LIN {X 0,Y 498.54,Z 668.142,A -85,B 0,C 180,E1 -12477.451,E2 -12477.451} C_VEL
LIN {X 0,Y 496.811,Z 689.973,A -85,B 0,C 180,E1 -12478.358,E2 -12478.358} C_VEL
LIN {X 0,Y 494.724,Z 710.777,A -85,B 0,C 180,E1 -12479.449,E2 -12479.449} C_VEL
LIN {X 0,Y 492.444,Z 730.313,A -85,B 0,C 180,E1 -12480.703,E2 -12480.703} C_VEL
LIN {X 0,Y 489.968,Z 749.027,A -85,B 0,C 180,E1 -12482.139,E2 -12482.139} C_VEL
LIN {X 0,Y 487.302,Z 767.508,A -85,B 0,C 180,E1 -12483.822,E2 -12483.822} C_VEL
LIN {X 0,Y 484.655,Z 784.843,A -85,B 0,C 180,E1 -12485.695,E2 -12485.695} C_VEL
LIN {X 0,Y 482.176,Z 800.537,A -85,B 0,C 180,E1 -12487.698,E2 -12487.698} C_VEL
LIN {X 0,Y 479.994,Z 814.356,A -85,B 0,C 180,E1 -12489.769,E2 -12489.769} C_VEL
LIN {X 0,Y 478.09,Z 826.817,A -85,B 0,C 180,E1 -12491.969,E2 -12491.969} C_VEL
LIN {X 0,Y 476.381,Z 838.536,A -85,B 0,C 180,E1 -12494.454,E2 -12494.454} C_VEL
LIN {X 0,Y 475.075,Z 848.28,A -85,B 0,C 180,E1 -12496.985,E2 -12496.985} C_VEL
LIN {X 0,Y 474.193,Z 855.818,A -85,B 0,C 180,E1 -12499.429,E2 -12499.429} C_VEL
LIN {X 0,Y 473.59,Z 861.948,A -85,B 0,C 180,E1 -12501.99,E2 -12501.99} C_VEL
LIN {X 0,Y 473.251,Z 866.357,A -85,B 0,C 180,E1 -12504.544,E2 -12504.544} C_VEL
LIN {X 0,Y 473.077,Z 869.113,A -85,B 0,C 180,E1 -12507.092,E2 -12507.092} C_VEL
LIN {X 0,Y 473.009,Z 870.147,A -85,B 0,C 180,E1 -12509.637,E2 -12509.637} C_VEL
LIN {X 0,Y 473.046,Z 869.578,A -85,B 0,C 180,E1 -12512.18,E2 -12512.18} C_VEL
LIN {X 0,Y 473.186,Z 867.412,A -85,B 0,C 180,E1 -12514.727,E2 -12514.727} C_VEL
LIN {X 0,Y 473.468,Z 863.613,A -85,B 0,C 180,E1 -12517.279,E2 -12517.279} C_VEL
LIN {X 0,Y 473.968,Z 858.017,A -85,B 0,C 180,E1 -12519.839,E2 -12519.839} C_VEL
LIN {X 0,Y 474.756,Z 851.005,A -85,B 0,C 180,E1 -12522.282,E2 -12522.282} C_VEL
LIN {X 0,Y 475.921,Z 841.751,A -85,B 0,C 180,E1 -12524.852,E2 -12524.852} C_VEL
LIN {X 0,Y 477.437,Z 831.152,A -85,B 0,C 180,E1 -12527.254,E2 -12527.254} C_VEL
LIN {X 0,Y 479.248,Z 819.296,A -85,B 0,C 180,E1 -12529.501,E2 -12529.501} C_VEL
LIN {X 0,Y 481.426,Z 805.537,A -85,B 0,C 180,E1 -12531.697,E2 -12531.697} C_VEL
LIN {X 0,Y 483.853,Z 790.18,A -85,B 0,C 180,E1 -12533.764,E2 -12533.764} C_VEL
LIN {X 0,Y 486.381,Z 773.879,A -85,B 0,C 180,E1 -12535.625,E2 -12535.625} C_VEL
LIN {X 0,Y 488.969,Z 756.338,A -85,B 0,C 180,E1 -12537.328,E2 -12537.328} C_VEL
LIN {X 0,Y 491.47,Z 738.084,A -85,B 0,C 180,E1 -12538.827,E2 -12538.827} C_VEL
LIN {X 0,Y 493.925,Z 718.094,A -85,B 0,C 180,E1 -12540.202,E2 -12540.202} C_VEL
LIN {X 0,Y 496.061,Z 698.144,A -85,B 0,C 180,E1 -12541.335,E2 -12541.335} C_VEL
LIN {X 0,Y 497.882,Z 677.418,A -85,B 0,C 180,E1 -12542.29,E2 -12542.29} C_VEL
LIN {X 0,Y 499.402,Z 655.167,A -85,B 0,C 180,E1 -12543.082,E2 -12543.082} C_VEL
LIN {X 0,Y 501.293,Z 619.373,A -85,B 0,C 180,E1 -12543.999,E2 -12543.999} C_VEL
LIN {X 0,Y 506.162,Z 544.365,A -85,B 0,C 180,E1 -12545.618,E2 -12545.618} C_VEL
LIN {X 0,Y 509.917,Z 475.713,A -85,B 0,C 180,E1 -12546.907,E2 -12546.907} C_VEL
LIN {X 0,Y 512.618,Z 409.2,A -85,B 0,C 180,E1 -12547.977,E2 -12547.977} C_VEL
LIN {X 0,Y 513.876,Z 374.612,A -85,B 0,C 180,E1 -12548.51,E2 -12548.51} C_VEL
LIN {X 0,Y 517.445,Z 358.291,A -85,B 0,C 180,E1 -12549.153,E2 -12549.153} C_VEL
LIN {X 0,Y 517.911,Z 317.946,A -85,B 0,C 180,E1 -12551.929,E2 -12551.929} C_VEL
LIN {X 0,Y 510.317,Z 297.328,A -85,B 0,C 180,E1 -12554.386,E2 -12554.386} C_VEL
LIN {X 0,Y 502.334,Z 278.601,A -85,B 0,C 180,E1 -12556.785,E2 -12556.785} C_VEL
LIN {X 0,Y 494.836,Z 263.053,A -85,B 0,C 180,E1 -12558.95,E2 -12558.95} C_VEL
LIN {X 0,Y 487.309,Z 249.107,A -85,B 0,C 180,E1 -12561.046,E2 -12561.046} C_VEL
LIN {X 0,Y 482.169,Z 240.332,A -85,B 0,C 180,E1 -12562.434,E2 -12562.434} C_VEL
LIN {X 0,Y 479.749,Z 236.125,A -85,B 0,C 180,E1 -12563.112,E2 -12563.112} C_VEL
LIN {X 0,Y 477.498,Z 232.436,A -85,B 0,C 180,E1 -12563.726,E2 -12563.726} C_VEL
LIN {X 0,Y 476.91,Z 231.296,A -85,B 0,C 180,E1 -12563.903,E2 -12563.903} C_VEL
LIN {X 0,Y 474.742,Z 228.427,A -85,B 0,C 180,E1 -12564.457,E2 -12564.457} C_VEL
LIN {X 0,Y 474.109,Z 226.17,A -85,B 0,C 180,E1 -12564.742,E2 -12564.742} C_VEL
LIN {X 0,Y 474.113,Z 226.159,A -85,B 0,C 180,E1 -12568.464,E2 -12568.464} C_VEL
LIN {X 0,Y 474.107,Z 226.143,A -85,B 0,C 180,E1 -12572.088,E2 -12572.088} C_VEL
LIN {X 0,Y 474.108,Z 226.139,A -85,B 0,C 180,E1 -12575.716,E2 -12575.716} C_VEL
LIN {X 0,Y 474.107,Z 226.173,A -85,B 0,C 180,E1 -12579.378,E2 -12579.378} C_VEL
LIN {X 0,Y 474.105,Z 226.141,A -85,B 0,C 180,E1 -12583.08,E2 -12583.08} C_VEL
LIN {X 0,Y 474.101,Z 226.141,A -85,B 0,C 180,E1 -12586.585,E2 -12586.585} C_VEL
LIN {X 0,Y 474.099,Z 226.17,A -85,B 0,C 180,E1 -12590.286,E2 -12590.286} C_VEL
LIN {X 0,Y 474.103,Z 226.127,A -85,B 0,C 180,E1 -12593.947,E2 -12593.947} C_VEL
LIN {X 0,Y 474.112,Z 226.175,A -85,B 0,C 180,E1 -12597.583,E2 -12597.583} C_VEL
LIN {X 0,Y 474.109,Z 226.126,A -85,B 0,C 180,E1 -12601.208,E2 -12601.208} C_VEL
LIN {X 0,Y 474.1,Z 226.168,A -85,B 0,C 180,E1 -12604.839,E2 -12604.839} C_VEL
LIN {X 0,Y 474.084,Z 226.14,A -85,B 0,C 180,E1 -12608.441,E2 -12608.441} C_VEL
LIN {X 0,Y 474.099,Z 226.178,A -85,B 0,C 180,E1 -12612.052,E2 -12612.052} C_VEL
LIN {X 0,Y 474.117,Z 226.162,A -85,B 0,C 180,E1 -12615.661,E2 -12615.661} C_VEL
LIN {X 0,Y 474.116,Z 226.167,A -85,B 0,C 180,E1 -12619.336,E2 -12619.336} C_VEL
LIN {X 0,Y 474.086,Z 226.178,A -85,B 0,C 180,E1 -12622.835,E2 -12622.835} C_VEL
LIN {X 0,Y 474.083,Z 226.168,A -85,B 0,C 180,E1 -12626.425,E2 -12626.425} C_VEL
LIN {X 0,Y 474.134,Z 226.296,A -85,B 0,C 180,E1 -12627.45,E2 -12627.45} C_VEL
LIN {X 0,Y 475.326,Z 229.528,A -85,B 0,C 180,E1 -12627.976,E2 -12627.976} C_VEL
LIN {X 0,Y 476.699,Z 231.84,A -85,B 0,C 180,E1 -12628.434,E2 -12628.434} C_VEL
LIN {X 0,Y 481.647,Z 241.457,A -85,B 0,C 180,E1 -12630.158,E2 -12630.158} C_VEL
LIN {X 0,Y 489.624,Z 256.766,A -85,B 0,C 180,E1 -12632.764,E2 -12632.764} C_VEL
LIN {X 0,Y 500.094,Z 277.627,A -85,B 0,C 180,E1 -12636.003,E2 -12636.003} C_VEL
LIN {X 0,Y 511.483,Z 301.22,A -85,B 0,C 180,E1 -12639.3,E2 -12639.3} C_VEL
LIN {X 0,Y 519.807,Z 318.56,A -85,B 0,C 180,E1 -12641.486,E2 -12641.486} C_VEL
LIN {X 0,Y 522.352,Z 322.995,A -85,B 0,C 180,E1 -12641.812,E2 -12641.812} C_VEL
LIN {X 0,Y 524.642,Z 347.742,A -85,B 0,C 180,E1 -12642.536,E2 -12642.536} C_VEL
LIN {X 0,Y 513.943,Z 587.488,A -85,B 0,C 180,E1 -12646.538,E2 -12646.538} C_VEL
LIN {X 0,Y 509.832,Z 692.964,A -85,B 0,C 180,E1 -12648.278,E2 -12648.278} C_VEL
LIN {X 0,Y 508.032,Z 717.442,A -85,B 0,C 180,E1 -12648.868,E2 -12648.868} C_VEL
LIN {X 0,Y 505.864,Z 741.406,A -85,B 0,C 180,E1 -12649.63,E2 -12649.63} C_VEL
LIN {X 0,Y 503.324,Z 764.227,A -85,B 0,C 180,E1 -12650.565,E2 -12650.565} C_VEL
LIN {X 0,Y 500.285,Z 788.254,A -85,B 0,C 180,E1 -12651.764,E2 -12651.764} C_VEL
LIN {X 0,Y 497.424,Z 808.594,A -85,B 0,C 180,E1 -12652.984,E2 -12652.984} C_VEL
LIN {X 0,Y 493.885,Z 831.697,A -85,B 0,C 180,E1 -12654.618,E2 -12654.618} C_VEL
LIN {X 0,Y 490.913,Z 850.192,A -85,B 0,C 180,E1 -12656.147,E2 -12656.147} C_VEL
LIN {X 0,Y 487.599,Z 870.092,A -85,B 0,C 180,E1 -12658.058,E2 -12658.058} C_VEL
LIN {X 0,Y 484.649,Z 887.507,A -85,B 0,C 180,E1 -12659.98,E2 -12659.98} C_VEL
LIN {X 0,Y 481.773,Z 904.616,A -85,B 0,C 180,E1 -12662.162,E2 -12662.162} C_VEL
LIN {X 0,Y 479.426,Z 919.191,A -85,B 0,C 180,E1 -12664.291,E2 -12664.291} C_VEL
LIN {X 0,Y 477.164,Z 934.025,A -85,B 0,C 180,E1 -12666.799,E2 -12666.799} C_VEL
LIN {X 0,Y 475.501,Z 946.237,A -85,B 0,C 180,E1 -12669.184,E2 -12669.184} C_VEL
LIN {X 0,Y 474.103,Z 958.209,A -85,B 0,C 180,E1 -12671.939,E2 -12671.939} C_VEL
LIN {X 0,Y 473.22,Z 967.521,A -85,B 0,C 180,E1 -12674.474,E2 -12674.474} C_VEL
LIN {X 0,Y 472.64,Z 976.006,A -85,B 0,C 180,E1 -12677.29,E2 -12677.29} C_VEL
LIN {X 0,Y 472.385,Z 982.114,A -85,B 0,C 180,E1 -12679.822,E2 -12679.822} C_VEL
LIN {X 0,Y 472.289,Z 987.389,A -85,B 0,C 180,E1 -12682.702,E2 -12682.702} C_VEL
LIN {X 0,Y 472.333,Z 990.403,A -85,B 0,C 180,E1 -12685.143,E2 -12685.143} C_VEL
LIN {X 0,Y 472.382,Z 992.129,A -85,B 0,C 180,E1 -12687.452,E2 -12687.452} C_VEL
LIN {X 0,Y 472.425,Z 992.783,A -85,B 0,C 180,E1 -12690.121,E2 -12690.121} C_VEL
LIN {X 0,Y 472.4,Z 991.751,A -85,B 0,C 180,E1 -12692.79,E2 -12692.79} C_VEL
LIN {X 0,Y 472.366,Z 989.7,A -85,B 0,C 180,E1 -12695.101,E2 -12695.101} C_VEL
LIN {X 0,Y 472.343,Z 986.144,A -85,B 0,C 180,E1 -12697.664,E2 -12697.664} C_VEL
LIN {X 0,Y 472.457,Z 980.753,A -85,B 0,C 180,E1 -12700.364,E2 -12700.364} C_VEL
LIN {X 0,Y 472.711,Z 974.464,A -85,B 0,C 180,E1 -12702.832,E2 -12702.832} C_VEL
LIN {X 0,Y 473.282,Z 965.476,A -85,B 0,C 180,E1 -12705.689,E2 -12705.689} C_VEL
LIN {X 0,Y 474.142,Z 955.945,A -85,B 0,C 180,E1 -12708.186,E2 -12708.186} C_VEL
LIN {X 0,Y 475.522,Z 943.625,A -85,B 0,C 180,E1 -12710.945,E2 -12710.945} C_VEL
LIN {X 0,Y 477.241,Z 930.371,A -85,B 0,C 180,E1 -12713.458,E2 -12713.458} C_VEL
LIN {X 0,Y 479.545,Z 914.812,A -85,B 0,C 180,E1 -12716.016,E2 -12716.016} C_VEL
LIN {X 0,Y 482.006,Z 899.256,A -85,B 0,C 180,E1 -12718.227,E2 -12718.227} C_VEL
LIN {X 0,Y 485.194,Z 880.054,A -85,B 0,C 180,E1 -12720.599,E2 -12720.599} C_VEL
LIN {X 0,Y 488.36,Z 861.534,A -85,B 0,C 180,E1 -12722.58,E2 -12722.58} C_VEL
LIN {X 0,Y 491.865,Z 840.855,A -85,B 0,C 180,E1 -12724.481,E2 -12724.481} C_VEL
LIN {X 0,Y 495.389,Z 819.524,A -85,B 0,C 180,E1 -12726.177,E2 -12726.177} C_VEL
LIN {X 0,Y 498.74,Z 797.883,A -85,B 0,C 180,E1 -12727.635,E2 -12727.635} C_VEL
LIN {X 0,Y 502.253,Z 774.045,A -85,B 0,C 180,E1 -12728.984,E2 -12728.984} C_VEL
LIN {X 0,Y 505.228,Z 751.77,A -85,B 0,C 180,E1 -12730.031,E2 -12730.031} C_VEL
LIN {X 0,Y 507.919,Z 728.566,A -85,B 0,C 180,E1 -12730.907,E2 -12730.907} C_VEL
LIN {X 0,Y 510.279,Z 705.051,A -85,B 0,C 180,E1 -12731.608,E2 -12731.608} C_VEL
LIN {X 0,Y 512.094,Z 679.83,A -85,B 0,C 180,E1 -12732.154,E2 -12732.154} C_VEL
LIN {X 0,Y 517.017,Z 597.902,A -85,B 0,C 180,E1 -12733.672,E2 -12733.672} C_VEL
LIN {X 0,Y 522.642,Z 530.22,A -85,B 0,C 180,E1 -12735.047,E2 -12735.047} C_VEL
LIN {X 0,Y 529.867,Z 464.415,A -85,B 0,C 180,E1 -12736.492,E2 -12736.492} C_VEL
LIN {X 0,Y 538.765,Z 402.255,A -85,B 0,C 180,E1 -12737.913,E2 -12737.913} C_VEL
LIN {X 0,Y 544.168,Z 370.237,A -85,B 0,C 180,E1 -12738.674,E2 -12738.674} C_VEL
LIN {X 0,Y 538.418,Z 386.185,A -85,B 0,C 180,E1 -12740.242,E2 -12740.242} C_VEL
LIN {X 0,Y 534.921,Z 400.034,A -85,B 0,C 180,E1 -12741.47,E2 -12741.47} C_VEL
LIN {X 0,Y 531.61,Z 418.651,A -85,B 0,C 180,E1 -12742.928,E2 -12742.928} C_VEL
LIN {X 0,Y 528.747,Z 441.431,A -85,B 0,C 180,E1 -12744.455,E2 -12744.455} C_VEL
LIN {X 0,Y 526.309,Z 468.54,A -85,B 0,C 180,E1 -12746.028,E2 -12746.028} C_VEL
LIN {X 0,Y 524.021,Z 500.146,A -85,B 0,C 180,E1 -12747.6,E2 -12747.6} C_VEL
LIN {X 0,Y 523.085,Z 512.301,A -85,B 0,C 180,E1 -12748.121,E2 -12748.121} C_VEL
LIN {X 0,Y 507.968,Z 623.688,A -85,B 0,C 180,E1 -12751.162,E2 -12751.162} C_VEL
LIN {X 0,Y 500.211,Z 692.312,A -85,B 0,C 180,E1 -12753.095,E2 -12753.095} C_VEL
LIN {X 0,Y 497.222,Z 717.176,A -85,B 0,C 180,E1 -12754.031,E2 -12754.031} C_VEL
LIN {X 0,Y 494.515,Z 738.857,A -85,B 0,C 180,E1 -12755.066,E2 -12755.066} C_VEL
LIN {X 0,Y 491.751,Z 760.438,A -85,B 0,C 180,E1 -12756.323,E2 -12756.323} C_VEL
LIN {X 0,Y 489.036,Z 780.869,A -85,B 0,C 180,E1 -12757.774,E2 -12757.774} C_VEL
LIN {X 0,Y 486.605,Z 798.705,A -85,B 0,C 180,E1 -12759.303,E2 -12759.303} C_VEL
LIN {X 0,Y 484.482,Z 813.948,A -85,B 0,C 180,E1 -12760.843,E2 -12760.843} C_VEL
LIN {X 0,Y 482.34,Z 828.73,A -85,B 0,C 180,E1 -12762.632,E2 -12762.632} C_VEL
LIN {X 0,Y 480.502,Z 841.055,A -85,B 0,C 180,E1 -12764.428,E2 -12764.428} C_VEL
LIN {X 0,Y 478.852,Z 851.963,A -85,B 0,C 180,E1 -12766.352,E2 -12766.352} C_VEL
LIN {X 0,Y 477.393,Z 861.257,A -85,B 0,C 180,E1 -12768.4,E2 -12768.4} C_VEL
LIN {X 0,Y 476.233,Z 868.521,A -85,B 0,C 180,E1 -12770.452,E2 -12770.452} C_VEL
LIN {X 0,Y 475.29,Z 874.171,A -85,B 0,C 180,E1 -12772.627,E2 -12772.627} C_VEL
LIN {X 0,Y 474.594,Z 877.91,A -85,B 0,C 180,E1 -12774.802,E2 -12774.802} C_VEL
LIN {X 0,Y 474.097,Z 879.81,A -85,B 0,C 180,E1 -12776.978,E2 -12776.978} C_VEL
LIN {X 0,Y 473.788,Z 879.972,A -85,B 0,C 180,E1 -12779.033,E2 -12779.033} C_VEL
LIN {X 0,Y 473.605,Z 878.463,A -85,B 0,C 180,E1 -12781.21,E2 -12781.21} C_VEL
LIN {X 0,Y 473.549,Z 875.211,A -85,B 0,C 180,E1 -12783.389,E2 -12783.389} C_VEL
LIN {X 0,Y 473.645,Z 870.182,A -85,B 0,C 180,E1 -12785.573,E2 -12785.573} C_VEL
LIN {X 0,Y 473.915,Z 863.283,A -85,B 0,C 180,E1 -12787.76,E2 -12787.76} C_VEL
LIN {X 0,Y 474.405,Z 854.34,A -85,B 0,C 180,E1 -12789.952,E2 -12789.952} C_VEL
LIN {X 0,Y 475.124,Z 843.798,A -85,B 0,C 180,E1 -12792.025,E2 -12792.025} C_VEL
LIN {X 0,Y 476.057,Z 831.7,A -85,B 0,C 180,E1 -12793.983,E2 -12793.983} C_VEL
LIN {X 0,Y 477.184,Z 818.188,A -85,B 0,C 180,E1 -12795.807,E2 -12795.807} C_VEL
LIN {X 0,Y 478.539,Z 802.58,A -85,B 0,C 180,E1 -12797.574,E2 -12797.574} C_VEL
LIN {X 0,Y 480.003,Z 785.869,A -85,B 0,C 180,E1 -12799.153,E2 -12799.153} C_VEL
LIN {X 0,Y 481.552,Z 767.326,A -85,B 0,C 180,E1 -12800.607,E2 -12800.607} C_VEL
LIN {X 0,Y 483.066,Z 748.687,A -85,B 0,C 180,E1 -12801.811,E2 -12801.811} C_VEL
LIN {X 0,Y 484.603,Z 728.049,A -85,B 0,C 180,E1 -12802.888,E2 -12802.888} C_VEL
LIN {X 0,Y 486.002,Z 706.513,A -85,B 0,C 180,E1 -12803.764,E2 -12803.764} C_VEL
LIN {X 0,Y 487.201,Z 684.993,A -85,B 0,C 180,E1 -12804.407,E2 -12804.407} C_VEL
LIN {X 0,Y 491.38,Z 580.934,A -85,B 0,C 180,E1 -12806.484,E2 -12806.484} C_VEL
LIN {X 0,Y 494.767,Z 499.908,A -85,B 0,C 180,E1 -12808.079,E2 -12808.079} C_VEL
LIN {X 0,Y 489.856,Z 444.398,A -85,B 0,C 180,E1 -12809.669,E2 -12809.669} C_VEL
LIN {X 0,Y 494.577,Z 391.935,A -85,B 0,C 180,E1 -12813.597,E2 -12813.597} C_VEL
LIN {X 0,Y 499.626,Z 341.605,A -85,B 0,C 180,E1 -12817.391,E2 -12817.391} C_VEL
LIN {X 0,Y 504.089,Z 300.496,A -85,B 0,C 180,E1 -12820.518,E2 -12820.518} C_VEL
LIN {X 0,Y 497.077,Z 281.186,A -85,B 0,C 180,E1 -12822.836,E2 -12822.836} C_VEL
LIN {X 0,Y 498.864,Z 281.752,A -85,B 0,C 180,E1 -12823.116,E2 -12823.116} C_VEL
LIN {X 0,Y 503.777,Z 281.964,A -85,B 0,C 180,E1 -12823.765,E2 -12823.765} C_VEL
LIN {X 0,Y 511.406,Z 300.357,A -85,B 0,C 180,E1 -12826.095,E2 -12826.095} C_VEL
LIN {X 0,Y 517.83,Z 317.866,A -85,B 0,C 180,E1 -12828.168,E2 -12828.168} C_VEL
LIN {X 0,Y 517.363,Z 358.606,A -85,B 0,C 180,E1 -12830.97,E2 -12830.97} C_VEL
LIN {X 0,Y 513.648,Z 376.214,A -85,B 0,C 180,E1 -12831.628,E2 -12831.628} C_VEL
LIN {X 0,Y 510.519,Z 461.786,A -85,B 0,C 180,E1 -12832.95,E2 -12832.95} C_VEL
LIN {X 0,Y 507.289,Z 524.733,A -85,B 0,C 180,E1 -12834.092,E2 -12834.092} C_VEL
LIN {X 0,Y 506.039,Z 532.367,A -85,B 0,C 180,E1 -12834.17,E2 -12834.17} C_VEL
LIN {X 0,Y 499.793,Z 552.676,A -85,B 0,C 180,E1 -12834.148,E2 -12834.148} C_VEL
LIN {X 0,Y 498.777,Z 559.214,A -85,B 0,C 180,E1 -12834.234,E2 -12834.234} C_VEL
LIN {X 0,Y 493.831,Z 632.998,A -85,B 0,C 180,E1 -12835.9,E2 -12835.9} C_VEL
LIN {X 0,Y 492.338,Z 660.657,A -85,B 0,C 180,E1 -12836.672,E2 -12836.672} C_VEL
LIN {X 0,Y 490.752,Z 682.372,A -85,B 0,C 180,E1 -12837.494,E2 -12837.494} C_VEL
LIN {X 0,Y 488.846,Z 702.844,A -85,B 0,C 180,E1 -12838.481,E2 -12838.481} C_VEL
LIN {X 0,Y 486.522,Z 723.263,A -85,B 0,C 180,E1 -12839.699,E2 -12839.699} C_VEL
LIN {X 0,Y 483.983,Z 742.53,A -85,B 0,C 180,E1 -12841.09,E2 -12841.09} C_VEL
LIN {X 0,Y 481.322,Z 760.902,A -85,B 0,C 180,E1 -12842.671,E2 -12842.671} C_VEL
LIN {X 0,Y 478.596,Z 778.314,A -85,B 0,C 180,E1 -12844.442,E2 -12844.442} C_VEL
LIN {X 0,Y 476.006,Z 794.203,A -85,B 0,C 180,E1 -12846.346,E2 -12846.346} C_VEL
LIN {X 0,Y 473.532,Z 809.093,A -85,B 0,C 180,E1 -12848.444,E2 -12848.444} C_VEL
LIN {X 0,Y 471.329,Z 822.494,A -85,B 0,C 180,E1 -12850.674,E2 -12850.674} C_VEL
LIN {X 0,Y 469.449,Z 834.427,A -85,B 0,C 180,E1 -12853.034,E2 -12853.034} C_VEL
LIN {X 0,Y 467.909,Z 844.825,A -85,B 0,C 180,E1 -12855.521,E2 -12855.521} C_VEL
LIN {X 0,Y 466.793,Z 853.257,A -85,B 0,C 180,E1 -12858.008,E2 -12858.008} C_VEL
LIN {X 0,Y 466.006,Z 859.958,A -85,B 0,C 180,E1 -12860.49,E2 -12860.49} C_VEL
LIN {X 0,Y 465.509,Z 865.261,A -85,B 0,C 180,E1 -12863.091,E2 -12863.091} C_VEL
LIN {X 0,Y 465.23,Z 868.891,A -85,B 0,C 180,E1 -12865.686,E2 -12865.686} C_VEL
LIN {X 0,Y 465.099,Z 870.797,A -85,B 0,C 180,E1 -12868.275,E2 -12868.275} C_VEL
LIN {X 0,Y 465.069,Z 871.098,A -85,B 0,C 180,E1 -12870.739,E2 -12870.739} C_VEL
LIN {X 0,Y 465.149,Z 869.976,A -85,B 0,C 180,E1 -12873.204,E2 -12873.204} C_VEL
LIN {X 0,Y 465.356,Z 867.167,A -85,B 0,C 180,E1 -12875.796,E2 -12875.796} C_VEL
LIN {X 0,Y 465.713,Z 862.893,A -85,B 0,C 180,E1 -12878.271,E2 -12878.271} C_VEL
LIN {X 0,Y 466.373,Z 856.661,A -85,B 0,C 180,E1 -12880.904,E2 -12880.904} C_VEL
LIN {X 0,Y 467.313,Z 849.17,A -85,B 0,C 180,E1 -12883.361,E2 -12883.361} C_VEL
LIN {X 0,Y 468.657,Z 839.774,A -85,B 0,C 180,E1 -12885.848,E2 -12885.848} C_VEL
LIN {X 0,Y 470.425,Z 828.283,A -85,B 0,C 180,E1 -12888.335,E2 -12888.335} C_VEL
LIN {X 0,Y 472.548,Z 815.17,A -85,B 0,C 180,E1 -12890.693,E2 -12890.693} C_VEL
LIN {X 0,Y 474.847,Z 801.303,A -85,B 0,C 180,E1 -12892.796,E2 -12892.796} C_VEL
LIN {X 0,Y 477.37,Z 786.058,A -85,B 0,C 180,E1 -12894.766,E2 -12894.766} C_VEL
LIN {X 0,Y 480.042,Z 769.347,A -85,B 0,C 180,E1 -12896.604,E2 -12896.604} C_VEL
LIN {X 0,Y 482.71,Z 751.732,A -85,B 0,C 180,E1 -12898.25,E2 -12898.25} C_VEL
LIN {X 0,Y 485.282,Z 733.327,A -85,B 0,C 180,E1 -12899.705,E2 -12899.705} C_VEL
LIN {X 0,Y 487.727,Z 713.336,A -85,B 0,C 180,E1 -12901.024,E2 -12901.024} C_VEL
LIN {X 0,Y 489.988,Z 691.73,A -85,B 0,C 180,E1 -12902.182,E2 -12902.182} C_VEL
LIN {X 0,Y 491.801,Z 669.836,A -85,B 0,C 180,E1 -12903.107,E2 -12903.107} C_VEL
LIN {X 0,Y 493.107,Z 647.709,A -85,B 0,C 180,E1 -12903.816,E2 -12903.816} C_VEL
LIN {X 0,Y 495.899,Z 602.371,A -85,B 0,C 180,E1 -12904.921,E2 -12904.921} C_VEL
LIN {X 0,Y 500.552,Z 531.774,A -85,B 0,C 180,E1 -12906.421,E2 -12906.421} C_VEL
LIN {X 0,Y 504.112,Z 465.945,A -85,B 0,C 180,E1 -12907.639,E2 -12907.639} C_VEL
LIN {X 0,Y 507.201,Z 385.645,A -85,B 0,C 180,E1 -12908.901,E2 -12908.901} C_VEL
LIN {X 0,Y 507.596,Z 377.376,A -85,B 0,C 180,E1 -12909.04,E2 -12909.04} C_VEL
LIN {X 0,Y 511.408,Z 359.689,A -85,B 0,C 180,E1 -12909.743,E2 -12909.743} C_VEL
LIN {X 0,Y 511.798,Z 321.583,A -85,B 0,C 180,E1 -12912.378,E2 -12912.378} C_VEL
LIN {X 0,Y 503.702,Z 299.721,A -85,B 0,C 180,E1 -12915.033,E2 -12915.033} C_VEL
LIN {X 0,Y 495.259,Z 280.206,A -85,B 0,C 180,E1 -12917.598,E2 -12917.598} C_VEL
LIN {X 0,Y 487.022,Z 263.522,A -85,B 0,C 180,E1 -12920.013,E2 -12920.013} C_VEL
LIN {X 0,Y 480.126,Z 251.024,A -85,B 0,C 180,E1 -12921.943,E2 -12921.943} C_VEL
LIN {X 0,Y 474.875,Z 242.046,A -85,B 0,C 180,E1 -12923.424,E2 -12923.424} C_VEL
LIN {X 0,Y 472.072,Z 237.344,A -85,B 0,C 180,E1 -12924.226,E2 -12924.226} C_VEL
LIN {X 0,Y 469.994,Z 234.244,A -85,B 0,C 180,E1 -12924.792,E2 -12924.792} C_VEL
LIN {X 0,Y 469.308,Z 232.581,A -85,B 0,C 180,E1 -12925.032,E2 -12925.032} C_VEL
LIN {X 0,Y 467.108,Z 230.042,A -85,B 0,C 180,E1 -12925.589,E2 -12925.589} C_VEL
LIN {X 0,Y 466.171,Z 227.144,A -85,B 0,C 180,E1 -12925.994,E2 -12925.994} C_VEL
LIN {X 0,Y 466.183,Z 227.157,A -85,B 0,C 180,E1 -12929.732,E2 -12929.732} C_VEL
LIN {X 0,Y 466.167,Z 227.157,A -85,B 0,C 180,E1 -12933.435,E2 -12933.435} C_VEL
LIN {X 0,Y 466.163,Z 227.125,A -85,B 0,C 180,E1 -12937.155,E2 -12937.155} C_VEL
LIN {X 0,Y 466.169,Z 227.13,A -85,B 0,C 180,E1 -12940.712,E2 -12940.712} C_VEL
LIN {X 0,Y 466.166,Z 227.16,A -85,B 0,C 180,E1 -12944.448,E2 -12944.448} C_VEL
LIN {X 0,Y 466.157,Z 227.117,A -85,B 0,C 180,E1 -12948.117,E2 -12948.117} C_VEL
LIN {X 0,Y 466.173,Z 227.152,A -85,B 0,C 180,E1 -12951.737,E2 -12951.737} C_VEL
LIN {X 0,Y 466.167,Z 227.131,A -85,B 0,C 180,E1 -12955.448,E2 -12955.448} C_VEL
LIN {X 0,Y 466.172,Z 227.129,A -85,B 0,C 180,E1 -12959.14,E2 -12959.14} C_VEL
LIN {X 0,Y 466.16,Z 227.153,A -85,B 0,C 180,E1 -12962.828,E2 -12962.828} C_VEL
LIN {X 0,Y 466.145,Z 227.119,A -85,B 0,C 180,E1 -12966.404,E2 -12966.404} C_VEL
LIN {X 0,Y 466.16,Z 227.164,A -85,B 0,C 180,E1 -12970.09,E2 -12970.09} C_VEL
LIN {X 0,Y 466.178,Z 227.164,A -85,B 0,C 180,E1 -12973.773,E2 -12973.773} C_VEL
LIN {X 0,Y 466.178,Z 227.161,A -85,B 0,C 180,E1 -12977.475,E2 -12977.475} C_VEL
LIN {X 0,Y 466.164,Z 227.154,A -85,B 0,C 180,E1 -12981.122,E2 -12981.122} C_VEL
LIN {X 0,Y 466.143,Z 227.158,A -85,B 0,C 180,E1 -12984.726,E2 -12984.726} C_VEL
LIN {X 0,Y 466.167,Z 227.306,A -85,B 0,C 180,E1 -12986.359,E2 -12986.359} C_VEL
LIN {X 0,Y 467.547,Z 230.773,A -85,B 0,C 180,E1 -12986.961,E2 -12986.961} C_VEL
LIN {X 0,Y 468.637,Z 232.398,A -85,B 0,C 180,E1 -12987.305,E2 -12987.305} C_VEL
LIN {X 0,Y 470.585,Z 236.188,A -85,B 0,C 180,E1 -12988.007,E2 -12988.007} C_VEL
LIN {X 0,Y 479.969,Z 254.318,A -85,B 0,C 180,E1 -12991.247,E2 -12991.247} C_VEL
LIN {X 0,Y 490.555,Z 275.349,A -85,B 0,C 180,E1 -12994.659,E2 -12994.659} C_VEL
LIN {X 0,Y 500.946,Z 296.719,A -85,B 0,C 180,E1 -12997.791,E2 -12997.791} C_VEL
LIN {X 0,Y 511.695,Z 319.213,A -85,B 0,C 180,E1 -13000.761,E2 -13000.761} C_VEL
LIN {X 0,Y 516.358,Z 326.875,A -85,B 0,C 180,E1 -13001.352,E2 -13001.352} C_VEL
LIN {X 0,Y 518.336,Z 348.872,A -85,B 0,C 180,E1 -13002.004,E2 -13002.004} C_VEL
LIN {X 0,Y 507.238,Z 586.374,A -85,B 0,C 180,E1 -13006.036,E2 -13006.036} C_VEL
LIN {X 0,Y 502.902,Z 692.911,A -85,B 0,C 180,E1 -13007.824,E2 -13007.824} C_VEL
LIN {X 0,Y 501.042,Z 717.485,A -85,B 0,C 180,E1 -13008.425,E2 -13008.425} C_VEL
LIN {X 0,Y 498.81,Z 741.363,A -85,B 0,C 180,E1 -13009.195,E2 -13009.195} C_VEL
LIN {X 0,Y 496.263,Z 763.656,A -85,B 0,C 180,E1 -13010.117,E2 -13010.117} C_VEL
LIN {X 0,Y 493.243,Z 787.052,A -85,B 0,C 180,E1 -13011.29,E2 -13011.29} C_VEL
LIN {X 0,Y 490.284,Z 807.507,A -85,B 0,C 180,E1 -13012.525,E2 -13012.525} C_VEL
LIN {X 0,Y 486.843,Z 829.512,A -85,B 0,C 180,E1 -13014.085,E2 -13014.085} C_VEL
LIN {X 0,Y 483.717,Z 848.3,A -85,B 0,C 180,E1 -13015.645,E2 -13015.645} C_VEL
LIN {X 0,Y 480.169,Z 869.073,A -85,B 0,C 180,E1 -13017.645,E2 -13017.645} C_VEL
LIN {X 0,Y 477.21,Z 886.031,A -85,B 0,C 180,E1 -13019.532,E2 -13019.532} C_VEL
LIN {X 0,Y 474.101,Z 903.893,A -85,B 0,C 180,E1 -13021.833,E2 -13021.833} C_VEL
LIN {X 0,Y 471.568,Z 919.187,A -85,B 0,C 180,E1 -13024.101,E2 -13024.101} C_VEL
LIN {X 0,Y 469.349,Z 933.266,A -85,B 0,C 180,E1 -13026.523,E2 -13026.523} C_VEL
LIN {X 0,Y 467.629,Z 945.482,A -85,B 0,C 180,E1 -13028.948,E2 -13028.948} C_VEL
LIN {X 0,Y 466.173,Z 957.477,A -85,B 0,C 180,E1 -13031.751,E2 -13031.751} C_VEL
LIN {X 0,Y 465.263,Z 966.781,A -85,B 0,C 180,E1 -13034.322,E2 -13034.322} C_VEL
LIN {X 0,Y 464.669,Z 975.278,A -85,B 0,C 180,E1 -13037.195,E2 -13037.195} C_VEL
LIN {X 0,Y 464.416,Z 981.244,A -85,B 0,C 180,E1 -13039.714,E2 -13039.714} C_VEL
LIN {X 0,Y 464.32,Z 986.433,A -85,B 0,C 180,E1 -13042.576,E2 -13042.576} C_VEL
LIN {X 0,Y 464.373,Z 989.471,A -85,B 0,C 180,E1 -13045.059,E2 -13045.059} C_VEL
LIN {X 0,Y 464.429,Z 991.213,A -85,B 0,C 180,E1 -13047.409,E2 -13047.409} C_VEL
LIN {X 0,Y 464.477,Z 991.875,A -85,B 0,C 180,E1 -13050.123,E2 -13050.123} C_VEL
LIN {X 0,Y 464.447,Z 990.846,A -85,B 0,C 180,E1 -13052.838,E2 -13052.838} C_VEL
LIN {X 0,Y 464.405,Z 988.778,A -85,B 0,C 180,E1 -13055.188,E2 -13055.188} C_VEL
LIN {X 0,Y 464.382,Z 985.207,A -85,B 0,C 180,E1 -13057.796,E2 -13057.796} C_VEL
LIN {X 0,Y 464.483,Z 979.801,A -85,B 0,C 180,E1 -13060.543,E2 -13060.543} C_VEL
LIN {X 0,Y 464.771,Z 973.134,A -85,B 0,C 180,E1 -13063.182,E2 -13063.182} C_VEL
LIN {X 0,Y 465.389,Z 964.01,A -85,B 0,C 180,E1 -13066.091,E2 -13066.091} C_VEL
LIN {X 0,Y 466.305,Z 954.396,A -85,B 0,C 180,E1 -13068.633,E2 -13068.633} C_VEL
LIN {X 0,Y 467.802,Z 941.928,A -85,B 0,C 180,E1 -13071.438,E2 -13071.438} C_VEL
LIN {X 0,Y 469.561,Z 929.295,A -85,B 0,C 180,E1 -13073.865,E2 -13073.865} C_VEL
LIN {X 0,Y 471.941,Z 914.029,A -85,B 0,C 180,E1 -13076.418,E2 -13076.418} C_VEL
LIN {X 0,Y 474.607,Z 898.182,A -85,B 0,C 180,E1 -13078.708,E2 -13078.708} C_VEL
LIN {X 0,Y 477.963,Z 879.004,A -85,B 0,C 180,E1 -13081.113,E2 -13081.113} C_VEL
LIN {X 0,Y 481.406,Z 860.028,A -85,B 0,C 180,E1 -13083.171,E2 -13083.171} C_VEL
LIN {X 0,Y 485.017,Z 839.842,A -85,B 0,C 180,E1 -13085.047,E2 -13085.047} C_VEL
LIN {X 0,Y 488.706,Z 818.705,A -85,B 0,C 180,E1 -13086.753,E2 -13086.753} C_VEL
LIN {X 0,Y 492.221,Z 797.381,A -85,B 0,C 180,E1 -13088.211,E2 -13088.211} C_VEL
LIN {X 0,Y 495.94,Z 773.646,A -85,B 0,C 180,E1 -13089.576,E2 -13089.576} C_VEL
LIN {X 0,Y 499.069,Z 751.686,A -85,B 0,C 180,E1 -13090.628,E2 -13090.628} C_VEL
LIN {X 0,Y 501.964,Z 728.472,A -85,B 0,C 180,E1 -13091.523,E2 -13091.523} C_VEL
LIN {X 0,Y 504.399,Z 706.193,A -85,B 0,C 180,E1 -13092.208,E2 -13092.208} C_VEL
LIN {X 0,Y 506.382,Z 681.601,A -85,B 0,C 180,E1 -13092.767,E2 -13092.767} C_VEL
LIN {X 0,Y 511.96,Z 599.732,A -85,B 0,C 180,E1 -13094.343,E2 -13094.343} C_VEL
LIN {X 0,Y 518.163,Z 533.367,A -85,B 0,C 180,E1 -13095.738,E2 -13095.738} C_VEL
LIN {X 0,Y 525.811,Z 470.913,A -85,B 0,C 180,E1 -13097.15,E2 -13097.15} C_VEL
LIN {X 0,Y 535.086,Z 411.727,A -85,B 0,C 180,E1 -13098.528,E2 -13098.528} C_VEL
LIN {X 0,Y 539.64,Z 386.423,A -85,B 0,C 180,E1 -13099.133,E2 -13099.133} C_VEL
LIN {X 0,Y 534.431,Z 402.446,A -85,B 0,C 180,E1 -13100.59,E2 -13100.59} C_VEL
LIN {X 0,Y 530.546,Z 419.16,A -85,B 0,C 180,E1 -13101.938,E2 -13101.938} C_VEL
LIN {X 0,Y 526.896,Z 440.675,A -85,B 0,C 180,E1 -13103.45,E2 -13103.45} C_VEL
LIN {X 0,Y 523.592,Z 467.503,A -85,B 0,C 180,E1 -13105.072,E2 -13105.072} C_VEL
LIN {X 0,Y 520.576,Z 498.689,A -85,B 0,C 180,E1 -13106.687,E2 -13106.687} C_VEL
LIN {X 0,Y 519.163,Z 513.949,A -85,B 0,C 180,E1 -13107.374,E2 -13107.374} C_VEL
LIN {X 0,Y 503.179,Z 623.523,A -85,B 0,C 180,E1 -13110.425,E2 -13110.425} C_VEL
LIN {X 0,Y 494.715,Z 692.559,A -85,B 0,C 180,E1 -13112.421,E2 -13112.421} C_VEL
LIN {X 0,Y 491.531,Z 716.722,A -85,B 0,C 180,E1 -13113.349,E2 -13113.349} C_VEL
LIN {X 0,Y 488.391,Z 739.771,A -85,B 0,C 180,E1 -13114.471,E2 -13114.471} C_VEL
LIN {X 0,Y 485.547,Z 760.078,A -85,B 0,C 180,E1 -13115.678,E2 -13115.678} C_VEL
LIN {X 0,Y 482.62,Z 780.56,A -85,B 0,C 180,E1 -13117.141,E2 -13117.141} C_VEL
LIN {X 0,Y 479.706,Z 800.352,A -85,B 0,C 180,E1 -13118.863,E2 -13118.863} C_VEL
LIN {X 0,Y 477.171,Z 816.917,A -85,B 0,C 180,E1 -13120.602,E2 -13120.602} C_VEL
LIN {X 0,Y 475.127,Z 830.018,A -85,B 0,C 180,E1 -13122.233,E2 -13122.233} C_VEL
LIN {X 0,Y 473.167,Z 842.333,A -85,B 0,C 180,E1 -13124.055,E2 -13124.055} C_VEL
LIN {X 0,Y 471.382,Z 853.157,A -85,B 0,C 180,E1 -13126.006,E2 -13126.006} C_VEL
LIN {X 0,Y 469.813,Z 862.453,A -85,B 0,C 180,E1 -13128.086,E2 -13128.086} C_VEL
LIN {X 0,Y 468.488,Z 870.052,A -85,B 0,C 180,E1 -13130.293,E2 -13130.293} C_VEL
LIN {X 0,Y 467.481,Z 875.602,A -85,B 0,C 180,E1 -13132.503,E2 -13132.503} C_VEL
LIN {X 0,Y 466.732,Z 879.228,A -85,B 0,C 180,E1 -13134.714,E2 -13134.714} C_VEL
LIN {X 0,Y 466.2,Z 881.03,A -85,B 0,C 180,E1 -13136.926,E2 -13136.926} C_VEL
LIN {X 0,Y 465.854,Z 881.048,A -85,B 0,C 180,E1 -13139.139,E2 -13139.139} C_VEL
LIN {X 0,Y 465.66,Z 879.31,A -85,B 0,C 180,E1 -13141.353,E2 -13141.353} C_VEL
LIN {X 0,Y 465.608,Z 875.845,A -85,B 0,C 180,E1 -13143.571,E2 -13143.571} C_VEL
LIN {X 0,Y 465.719,Z 870.596,A -85,B 0,C 180,E1 -13145.792,E2 -13145.792} C_VEL
LIN {X 0,Y 466.015,Z 863.458,A -85,B 0,C 180,E1 -13148.017,E2 -13148.017} C_VEL
LIN {X 0,Y 466.507,Z 854.813,A -85,B 0,C 180,E1 -13150.123,E2 -13150.123} C_VEL
LIN {X 0,Y 467.208,Z 844.805,A -85,B 0,C 180,E1 -13152.107,E2 -13152.107} C_VEL
LIN {X 0,Y 468.166,Z 832.719,A -85,B 0,C 180,E1 -13154.092,E2 -13154.092} C_VEL
LIN {X 0,Y 469.327,Z 819.151,A -85,B 0,C 180,E1 -13155.952,E2 -13155.952} C_VEL
LIN {X 0,Y 470.666,Z 804.108,A -85,B 0,C 180,E1 -13157.686,E2 -13157.686} C_VEL
LIN {X 0,Y 472.163,Z 787.528,A -85,B 0,C 180,E1 -13159.291,E2 -13159.291} C_VEL
LIN {X 0,Y 473.767,Z 769.076,A -85,B 0,C 180,E1 -13160.779,E2 -13160.779} C_VEL
LIN {X 0,Y 475.377,Z 749.813,A -85,B 0,C 180,E1 -13162.052,E2 -13162.052} C_VEL
LIN {X 0,Y 476.956,Z 729.338,A -85,B 0,C 180,E1 -13163.146,E2 -13163.146} C_VEL
LIN {X 0,Y 478.443,Z 707.237,A -85,B 0,C 180,E1 -13164.066,E2 -13164.066} C_VEL
LIN {X 0,Y 479.691,Z 685.63,A -85,B 0,C 180,E1 -13164.729,E2 -13164.729} C_VEL
LIN {X 0,Y 481.691,Z 636.241,A -85,B 0,C 180,E1 -13165.753,E2 -13165.753} C_VEL
LIN {X 0,Y 487.592,Z 500.852,A -85,B 0,C 180,E1 -13168.482,E2 -13168.482} C_VEL
LIN {X 0,Y 482.649,Z 443.526,A -85,B 0,C 180,E1 -13170.158,E2 -13170.158} C_VEL
LIN {X 0,Y 487.555,Z 391.321,A -85,B 0,C 180,E1 -13174.114,E2 -13174.114} C_VEL
LIN {X 0,Y 492.883,Z 340.388,A -85,B 0,C 180,E1 -13178.003,E2 -13178.003} C_VEL
LIN {X 0,Y 497.018,Z 303.388,A -85,B 0,C 180,E1 -13180.849,E2 -13180.849} C_VEL
LIN {X 0,Y 491.675,Z 288.4,A -85,B 0,C 180,E1 -13182.665,E2 -13182.665} C_VEL
LIN {X 0,Y 493.95,Z 288.989,A -85,B 0,C 180,E1 -13183.015,E2 -13183.015} C_VEL
LIN {X 0,Y 499.293,Z 289.309,A -85,B 0,C 180,E1 -13183.741,E2 -13183.741} C_VEL
LIN {X 0,Y 507.081,Z 308.783,A -85,B 0,C 180,E1 -13186.202,E2 -13186.202} C_VEL
LIN {X 0,Y 511.777,Z 322.105,A -85,B 0,C 180,E1 -13187.772,E2 -13187.772} C_VEL
LIN {X 0,Y 511.313,Z 360.22,A -85,B 0,C 180,E1 -13190.398,E2 -13190.398} C_VEL
LIN {X 0,Y 507.373,Z 378.886,A -85,B 0,C 180,E1 -13191.096,E2 -13191.096} C_VEL
LIN {X 0,Y 504.154,Z 463.908,A -85,B 0,C 180,E1 -13192.422,E2 -13192.422} C_VEL
LIN {X 0,Y 500.507,Z 531.887,A -85,B 0,C 180,E1 -13193.677,E2 -13193.677} C_VEL
LIN {X 0,Y 498.777,Z 559.214,A -85,B 0,C 180,E1 -13194.234,E2 -13194.234} C_VEL
LIN {X 0,Y 497.486,Z 566.831,A -85,B 0,C 180,E1 -13194.326,E2 -13194.326} C_VEL
LIN {X 0,Y 491.089,Z 587.097,A -85,B 0,C 180,E1 -13194.33,E2 -13194.33} C_VEL
LIN {X 0,Y 490.025,Z 593.617,A -85,B 0,C 180,E1 -13194.426,E2 -13194.426} C_VEL
LIN {X 0,Y 486.575,Z 645.419,A -85,B 0,C 180,E1 -13195.686,E2 -13195.686} C_VEL
LIN {X 0,Y 485.245,Z 667.881,A -85,B 0,C 180,E1 -13196.386,E2 -13196.386} C_VEL
LIN {X 0,Y 483.547,Z 688.635,A -85,B 0,C 180,E1 -13197.239,E2 -13197.239} C_VEL
LIN {X 0,Y 481.427,Z 709.184,A -85,B 0,C 180,E1 -13198.3,E2 -13198.3} C_VEL
LIN {X 0,Y 478.958,Z 729.358,A -85,B 0,C 180,E1 -13199.578,E2 -13199.578} C_VEL
LIN {X 0,Y 476.375,Z 747.976,A -85,B 0,C 180,E1 -13200.997,E2 -13200.997} C_VEL
LIN {X 0,Y 473.544,Z 766.359,A -85,B 0,C 180,E1 -13202.661,E2 -13202.661} C_VEL
LIN {X 0,Y 470.669,Z 783.837,A -85,B 0,C 180,E1 -13204.539,E2 -13204.539} C_VEL
LIN {X 0,Y 467.905,Z 799.872,A -85,B 0,C 180,E1 -13206.58,E2 -13206.58} C_VEL
LIN {X 0,Y 465.271,Z 814.963,A -85,B 0,C 180,E1 -13208.858,E2 -13208.858} C_VEL
LIN {X 0,Y 463.008,Z 828.125,A -85,B 0,C 180,E1 -13211.23,E2 -13211.23} C_VEL
LIN {X 0,Y 461.172,Z 839.251,A -85,B 0,C 180,E1 -13213.629,E2 -13213.629} C_VEL
LIN {X 0,Y 459.702,Z 848.945,A -85,B 0,C 180,E1 -13216.157,E2 -13216.157} C_VEL
LIN {X 0,Y 458.578,Z 857.298,A -85,B 0,C 180,E1 -13218.87,E2 -13218.87} C_VEL
LIN {X 0,Y 457.875,Z 863.459,A -85,B 0,C 180,E1 -13221.46,E2 -13221.46} C_VEL
LIN {X 0,Y 457.457,Z 868.051,A -85,B 0,C 180,E1 -13224.103,E2 -13224.103} C_VEL
LIN {X 0,Y 457.224,Z 870.89,A -85,B 0,C 180,E1 -13226.74,E2 -13226.74} C_VEL
LIN {X 0,Y 457.135,Z 872.082,A -85,B 0,C 180,E1 -13229.248,E2 -13229.248} C_VEL
LIN {X 0,Y 457.162,Z 871.849,A -85,B 0,C 180,E1 -13231.755,E2 -13231.755} C_VEL
LIN {X 0,Y 457.302,Z 869.964,A -85,B 0,C 180,E1 -13234.403,E2 -13234.403} C_VEL
LIN {X 0,Y 457.597,Z 866.416,A -85,B 0,C 180,E1 -13237.029,E2 -13237.029} C_VEL
LIN {X 0,Y 458.118,Z 861.185,A -85,B 0,C 180,E1 -13239.675,E2 -13239.675} C_VEL
LIN {X 0,Y 458.958,Z 854.552,A -85,B 0,C 180,E1 -13242.2,E2 -13242.2} C_VEL
LIN {X 0,Y 460.152,Z 846.045,A -85,B 0,C 180,E1 -13244.767,E2 -13244.767} C_VEL
LIN {X 0,Y 461.846,Z 835.297,A -85,B 0,C 180,E1 -13247.384,E2 -13247.384} C_VEL
LIN {X 0,Y 463.962,Z 822.671,A -85,B 0,C 180,E1 -13249.908,E2 -13249.908} C_VEL
LIN {X 0,Y 466.31,Z 809.091,A -85,B 0,C 180,E1 -13252.172,E2 -13252.172} C_VEL
LIN {X 0,Y 468.767,Z 794.94,A -85,B 0,C 180,E1 -13254.176,E2 -13254.176} C_VEL
LIN {X 0,Y 471.488,Z 778.982,A -85,B 0,C 180,E1 -13256.107,E2 -13256.107} C_VEL
LIN {X 0,Y 474.336,Z 761.484,A -85,B 0,C 180,E1 -13257.903,E2 -13257.903} C_VEL
LIN {X 0,Y 477.008,Z 743.797,A -85,B 0,C 180,E1 -13259.443,E2 -13259.443} C_VEL
LIN {X 0,Y 479.644,Z 724.54,A -85,B 0,C 180,E1 -13260.852,E2 -13260.852} C_VEL
LIN {X 0,Y 482.044,Z 704.365,A -85,B 0,C 180,E1 -13262.074,E2 -13262.074} C_VEL
LIN {X 0,Y 484.165,Z 682.397,A -85,B 0,C 180,E1 -13263.145,E2 -13263.145} C_VEL
LIN {X 0,Y 485.877,Z 659.344,A -85,B 0,C 180,E1 -13264.008,E2 -13264.008} C_VEL
LIN {X 0,Y 487.914,Z 623.727,A -85,B 0,C 180,E1 -13264.967,E2 -13264.967} C_VEL
LIN {X 0,Y 492.911,Z 552.333,A -85,B 0,C 180,E1 -13266.57,E2 -13266.57} C_VEL
LIN {X 0,Y 496.796,Z 487.533,A -85,B 0,C 180,E1 -13267.835,E2 -13267.835} C_VEL
LIN {X 0,Y 499.705,Z 423.65,A -85,B 0,C 180,E1 -13268.904,E2 -13268.904} C_VEL
LIN {X 0,Y 501.36,Z 380.151,A -85,B 0,C 180,E1 -13269.583,E2 -13269.583} C_VEL
LIN {X 0,Y 505.415,Z 361.597,A -85,B 0,C 180,E1 -13270.31,E2 -13270.31} C_VEL
LIN {X 0,Y 505.768,Z 325.409,A -85,B 0,C 180,E1 -13272.823,E2 -13272.823} C_VEL
LIN {X 0,Y 497.877,Z 304.182,A -85,B 0,C 180,E1 -13275.42,E2 -13275.42} C_VEL
LIN {X 0,Y 489.767,Z 285.201,A -85,B 0,C 180,E1 -13277.961,E2 -13277.961} C_VEL
LIN {X 0,Y 481.64,Z 268.543,A -85,B 0,C 180,E1 -13280.406,E2 -13280.406} C_VEL
LIN {X 0,Y 474.838,Z 256.177,A -85,B 0,C 180,E1 -13282.362,E2 -13282.362} C_VEL
LIN {X 0,Y 470.082,Z 247.938,A -85,B 0,C 180,E1 -13283.749,E2 -13283.749} C_VEL
LIN {X 0,Y 467.272,Z 243.314,A -85,B 0,C 180,E1 -13284.556,E2 -13284.556} C_VEL
LIN {X 0,Y 464.53,Z 238.712,A -85,B 0,C 180,E1 -13285.371,E2 -13285.371} C_VEL
LIN {X 0,Y 462.104,Z 235.133,A -85,B 0,C 180,E1 -13286.065,E2 -13286.065} C_VEL
LIN {X 0,Y 461.413,Z 233.57,A -85,B 0,C 180,E1 -13286.306,E2 -13286.306} C_VEL
LIN {X 0,Y 459.273,Z 231.197,A -85,B 0,C 180,E1 -13286.876,E2 -13286.876} C_VEL
LIN {X 0,Y 458.221,Z 228.122,A -85,B 0,C 180,E1 -13287.311,E2 -13287.311} C_VEL
LIN {X 0,Y 458.227,Z 228.119,A -85,B 0,C 180,E1 -13291.047,E2 -13291.047} C_VEL
LIN {X 0,Y 458.232,Z 228.139,A -85,B 0,C 180,E1 -13294.679,E2 -13294.679} C_VEL
LIN {X 0,Y 458.229,Z 228.136,A -85,B 0,C 180,E1 -13298.367,E2 -13298.367} C_VEL
LIN {X 0,Y 458.225,Z 228.105,A -85,B 0,C 180,E1 -13302.081,E2 -13302.081} C_VEL
LIN {X 0,Y 458.235,Z 228.133,A -85,B 0,C 180,E1 -13305.854,E2 -13305.854} C_VEL
LIN {X 0,Y 458.231,Z 228.13,A -85,B 0,C 180,E1 -13309.565,E2 -13309.565} C_VEL
LIN {X 0,Y 458.23,Z 228.107,A -85,B 0,C 180,E1 -13313.233,E2 -13313.233} C_VEL
LIN {X 0,Y 458.23,Z 228.15,A -85,B 0,C 180,E1 -13316.998,E2 -13316.998} C_VEL
LIN {X 0,Y 458.214,Z 228.1,A -85,B 0,C 180,E1 -13320.625,E2 -13320.625} C_VEL
LIN {X 0,Y 458.213,Z 228.15,A -85,B 0,C 180,E1 -13324.38,E2 -13324.38} C_VEL
LIN {X 0,Y 458.218,Z 228.106,A -85,B 0,C 180,E1 -13328.028,E2 -13328.028} C_VEL
LIN {X 0,Y 458.234,Z 228.151,A -85,B 0,C 180,E1 -13331.708,E2 -13331.708} C_VEL
LIN {X 0,Y 458.242,Z 228.138,A -85,B 0,C 180,E1 -13335.439,E2 -13335.439} C_VEL
LIN {X 0,Y 458.227,Z 228.143,A -85,B 0,C 180,E1 -13339.118,E2 -13339.118} C_VEL
LIN {X 0,Y 458.206,Z 228.157,A -85,B 0,C 180,E1 -13342.721,E2 -13342.721} C_VEL
LIN {X 0,Y 458.248,Z 228.309,A -85,B 0,C 180,E1 -13345.216,E2 -13345.216} C_VEL
LIN {X 0,Y 459.502,Z 231.574,A -85,B 0,C 180,E1 -13345.799,E2 -13345.799} C_VEL
LIN {X 0,Y 460.611,Z 233.05,A -85,B 0,C 180,E1 -13346.147,E2 -13346.147} C_VEL
LIN {X 0,Y 462.422,Z 236.877,A -85,B 0,C 180,E1 -13346.867,E2 -13346.867} C_VEL
LIN {X 0,Y 470.046,Z 251.38,A -85,B 0,C 180,E1 -13349.572,E2 -13349.572} C_VEL
LIN {X 0,Y 479.662,Z 270.434,A -85,B 0,C 180,E1 -13352.819,E2 -13352.819} C_VEL
LIN {X 0,Y 489.067,Z 289.421,A -85,B 0,C 180,E1 -13355.784,E2 -13355.784} C_VEL
LIN {X 0,Y 499.32,Z 310.731,A -85,B 0,C 180,E1 -13358.813,E2 -13358.813} C_VEL
LIN {X 0,Y 504.05,Z 320.505,A -85,B 0,C 180,E1 -13360.07,E2 -13360.07} C_VEL
LIN {X 0,Y 510.322,Z 330.764,A -85,B 0,C 180,E1 -13360.894,E2 -13360.894} C_VEL
LIN {X 0,Y 511.985,Z 350.164,A -85,B 0,C 180,E1 -13361.474,E2 -13361.474} C_VEL
LIN {X 0,Y 500.204,Z 594.045,A -85,B 0,C 180,E1 -13365.667,E2 -13365.667} C_VEL
LIN {X 0,Y 495.978,Z 693.246,A -85,B 0,C 180,E1 -13367.366,E2 -13367.366} C_VEL
LIN {X 0,Y 494.054,Z 717.678,A -85,B 0,C 180,E1 -13367.976,E2 -13367.976} C_VEL
LIN {X 0,Y 491.76,Z 741.384,A -85,B 0,C 180,E1 -13368.754,E2 -13368.754} C_VEL
LIN {X 0,Y 489.157,Z 763.478,A -85,B 0,C 180,E1 -13369.681,E2 -13369.681} C_VEL
LIN {X 0,Y 486.107,Z 786.461,A -85,B 0,C 180,E1 -13370.847,E2 -13370.847} C_VEL
LIN {X 0,Y 482.946,Z 807.676,A -85,B 0,C 180,E1 -13372.146,E2 -13372.146} C_VEL
LIN {X 0,Y 479.236,Z 830.66,A -85,B 0,C 180,E1 -13373.81,E2 -13373.81} C_VEL
LIN {X 0,Y 475.951,Z 849.917,A -85,B 0,C 180,E1 -13375.443,E2 -13375.443} C_VEL
LIN {X 0,Y 472.486,Z 869.477,A -85,B 0,C 180,E1 -13377.38,E2 -13377.38} C_VEL
LIN {X 0,Y 469.3,Z 887.249,A -85,B 0,C 180,E1 -13379.403,E2 -13379.403} C_VEL
LIN {X 0,Y 466.342,Z 903.708,A -85,B 0,C 180,E1 -13381.576,E2 -13381.576} C_VEL
LIN {X 0,Y 463.846,Z 918.314,A -85,B 0,C 180,E1 -13383.774,E2 -13383.774} C_VEL
LIN {X 0,Y 461.437,Z 933.109,A -85,B 0,C 180,E1 -13386.367,E2 -13386.367} C_VEL
LIN {X 0,Y 459.594,Z 945.92,A -85,B 0,C 180,E1 -13388.963,E2 -13388.963} C_VEL
LIN {X 0,Y 458.192,Z 957.214,A -85,B 0,C 180,E1 -13391.685,E2 -13391.685} C_VEL
LIN {X 0,Y 457.245,Z 966.776,A -85,B 0,C 180,E1 -13394.397,E2 -13394.397} C_VEL
LIN {X 0,Y 456.681,Z 974.841,A -85,B 0,C 180,E1 -13397.224,E2 -13397.224} C_VEL
LIN {X 0,Y 456.438,Z 980.733,A -85,B 0,C 180,E1 -13399.779,E2 -13399.779} C_VEL
LIN {X 0,Y 456.363,Z 985.805,A -85,B 0,C 180,E1 -13402.699,E2 -13402.699} C_VEL
LIN {X 0,Y 456.421,Z 988.645,A -85,B 0,C 180,E1 -13405.099,E2 -13405.099} C_VEL
LIN {X 0,Y 456.484,Z 990.35,A -85,B 0,C 180,E1 -13407.489,E2 -13407.489} C_VEL
LIN {X 0,Y 456.52,Z 990.948,A -85,B 0,C 180,E1 -13410.251,E2 -13410.251} C_VEL
LIN {X 0,Y 456.496,Z 989.935,A -85,B 0,C 180,E1 -13412.888,E2 -13412.888} C_VEL
LIN {X 0,Y 456.445,Z 987.861,A -85,B 0,C 180,E1 -13415.279,E2 -13415.279} C_VEL
LIN {X 0,Y 456.426,Z 984.128,A -85,B 0,C 180,E1 -13418.028,E2 -13418.028} C_VEL
LIN {X 0,Y 456.512,Z 978.559,A -85,B 0,C 180,E1 -13420.857,E2 -13420.857} C_VEL
LIN {X 0,Y 456.806,Z 972.154,A -85,B 0,C 180,E1 -13423.416,E2 -13423.416} C_VEL
LIN {X 0,Y 457.471,Z 963.024,A -85,B 0,C 180,E1 -13426.377,E2 -13426.377} C_VEL
LIN {X 0,Y 458.432,Z 953.388,A -85,B 0,C 180,E1 -13428.965,E2 -13428.965} C_VEL
LIN {X 0,Y 460.047,Z 940.686,A -85,B 0,C 180,E1 -13431.864,E2 -13431.864} C_VEL
LIN {X 0,Y 461.929,Z 928.114,A -85,B 0,C 180,E1 -13434.314,E2 -13434.314} C_VEL
LIN {X 0,Y 464.561,Z 912.168,A -85,B 0,C 180,E1 -13437.01,E2 -13437.01} C_VEL
LIN {X 0,Y 467.24,Z 897.186,A -85,B 0,C 180,E1 -13439.204,E2 -13439.204} C_VEL
LIN {X 0,Y 470.791,Z 878.062,A -85,B 0,C 180,E1 -13441.641,E2 -13441.641} C_VEL
LIN {X 0,Y 474.441,Z 859.063,A -85,B 0,C 180,E1 -13443.734,E2 -13443.734} C_VEL
LIN {X 0,Y 478.199,Z 839.149,A -85,B 0,C 180,E1 -13445.615,E2 -13445.615} C_VEL
LIN {X 0,Y 482.12,Z 818.027,A -85,B 0,C 180,E1 -13447.346,E2 -13447.346} C_VEL
LIN {X 0,Y 485.785,Z 797.142,A -85,B 0,C 180,E1 -13448.798,E2 -13448.798} C_VEL
LIN {X 0,Y 489.724,Z 773.628,A -85,B 0,C 180,E1 -13450.18,E2 -13450.18} C_VEL
LIN {X 0,Y 493.009,Z 752.05,A -85,B 0,C 180,E1 -13451.235,E2 -13451.235} C_VEL
LIN {X 0,Y 496.262,Z 727.875,A -85,B 0,C 180,E1 -13452.189,E2 -13452.189} C_VEL
LIN {X 0,Y 498.951,Z 704.878,A -85,B 0,C 180,E1 -13452.906,E2 -13452.906} C_VEL
LIN {X 0,Y 501.206,Z 679.012,A -85,B 0,C 180,E1 -13453.498,E2 -13453.498} C_VEL
LIN {X 0,Y 506.91,Z 604.456,A -85,B 0,C 180,E1 -13454.984,E2 -13454.984} C_VEL
LIN {X 0,Y 513.515,Z 540.682,A -85,B 0,C 180,E1 -13456.364,E2 -13456.364} C_VEL
LIN {X 0,Y 521.895,Z 478.411,A -85,B 0,C 180,E1 -13457.804,E2 -13457.804} C_VEL
LIN {X 0,Y 532.261,Z 418.01,A -85,B 0,C 180,E1 -13459.232,E2 -13459.232} C_VEL
LIN {X 0,Y 535.068,Z 403.51,A -85,B 0,C 180,E1 -13459.593,E2 -13459.593} C_VEL
LIN {X 0,Y 529.965,Z 420.849,A -85,B 0,C 180,E1 -13461.024,E2 -13461.024} C_VEL
LIN {X 0,Y 525.36,Z 442.234,A -85,B 0,C 180,E1 -13462.56,E2 -13462.56} C_VEL
LIN {X 0,Y 521.359,Z 467.462,A -85,B 0,C 180,E1 -13464.133,E2 -13464.133} C_VEL
LIN {X 0,Y 517.712,Z 496.915,A -85,B 0,C 180,E1 -13465.72,E2 -13465.72} C_VEL
LIN {X 0,Y 515.606,Z 515.721,A -85,B 0,C 180,E1 -13466.602,E2 -13466.602} C_VEL
LIN {X 0,Y 498.716,Z 623.519,A -85,B 0,C 180,E1 -13469.657,E2 -13469.657} C_VEL
LIN {X 0,Y 489.462,Z 693.045,A -85,B 0,C 180,E1 -13471.718,E2 -13471.718} C_VEL
LIN {X 0,Y 485.921,Z 717.566,A -85,B 0,C 180,E1 -13472.686,E2 -13472.686} C_VEL
LIN {X 0,Y 482.406,Z 741.177,A -85,B 0,C 180,E1 -13473.867,E2 -13473.867} C_VEL
LIN {X 0,Y 479.01,Z 763.375,A -85,B 0,C 180,E1 -13475.234,E2 -13475.234} C_VEL
LIN {X 0,Y 475.96,Z 782.652,A -85,B 0,C 180,E1 -13476.672,E2 -13476.672} C_VEL
LIN {X 0,Y 473.172,Z 800.284,A -85,B 0,C 180,E1 -13478.231,E2 -13478.231} C_VEL
LIN {X 0,Y 470.431,Z 816.956,A -85,B 0,C 180,E1 -13479.989,E2 -13479.989} C_VEL
LIN {X 0,Y 467.973,Z 831.456,A -85,B 0,C 180,E1 -13481.823,E2 -13481.823} C_VEL
LIN {X 0,Y 465.858,Z 843.626,A -85,B 0,C 180,E1 -13483.67,E2 -13483.67} C_VEL
LIN {X 0,Y 463.953,Z 854.446,A -85,B 0,C 180,E1 -13485.65,E2 -13485.65} C_VEL
LIN {X 0,Y 462.258,Z 863.686,A -85,B 0,C 180,E1 -13487.762,E2 -13487.762} C_VEL
LIN {X 0,Y 460.893,Z 870.899,A -85,B 0,C 180,E1 -13489.879,E2 -13489.879} C_VEL
LIN {X 0,Y 459.777,Z 876.529,A -85,B 0,C 180,E1 -13492.125,E2 -13492.125} C_VEL
LIN {X 0,Y 458.985,Z 880.06,A -85,B 0,C 180,E1 -13494.249,E2 -13494.249} C_VEL
LIN {X 0,Y 458.376,Z 882.037,A -85,B 0,C 180,E1 -13496.498,E2 -13496.498} C_VEL
LIN {X 0,Y 457.98,Z 882.254,A -85,B 0,C 180,E1 -13498.749,E2 -13498.749} C_VEL
LIN {X 0,Y 457.742,Z 880.699,A -85,B 0,C 180,E1 -13501.001,E2 -13501.001} C_VEL
LIN {X 0,Y 457.661,Z 877.402,A -85,B 0,C 180,E1 -13503.256,E2 -13503.256} C_VEL
LIN {X 0,Y 457.746,Z 872.332,A -85,B 0,C 180,E1 -13505.515,E2 -13505.515} C_VEL
LIN {X 0,Y 458.022,Z 865.378,A -85,B 0,C 180,E1 -13507.779,E2 -13507.779} C_VEL
LIN {X 0,Y 458.534,Z 856.372,A -85,B 0,C 180,E1 -13510.047,E2 -13510.047} C_VEL
LIN {X 0,Y 459.29,Z 845.771,A -85,B 0,C 180,E1 -13512.191,E2 -13512.191} C_VEL
LIN {X 0,Y 460.275,Z 833.663,A -85,B 0,C 180,E1 -13514.21,E2 -13514.21} C_VEL
LIN {X 0,Y 461.471,Z 820.087,A -85,B 0,C 180,E1 -13516.102,E2 -13516.102} C_VEL
LIN {X 0,Y 462.908,Z 804.481,A -85,B 0,C 180,E1 -13517.927,E2 -13517.927} C_VEL
LIN {X 0,Y 464.458,Z 787.813,A -85,B 0,C 180,E1 -13519.558,E2 -13519.558} C_VEL
LIN {X 0,Y 466.117,Z 769.248,A -85,B 0,C 180,E1 -13521.07,E2 -13521.07} C_VEL
LIN {X 0,Y 467.783,Z 749.889,A -85,B 0,C 180,E1 -13522.363,E2 -13522.363} C_VEL
LIN {X 0,Y 469.412,Z 729.333,A -85,B 0,C 180,E1 -13523.474,E2 -13523.474} C_VEL
LIN {X 0,Y 470.946,Z 707.195,A -85,B 0,C 180,E1 -13524.407,E2 -13524.407} C_VEL
LIN {X 0,Y 472.25,Z 685.306,A -85,B 0,C 180,E1 -13525.087,E2 -13525.087} C_VEL
LIN {X 0,Y 476.139,Z 594.578,A -85,B 0,C 180,E1 -13526.978,E2 -13526.978} C_VEL
LIN {X 0,Y 480.399,Z 501.629,A -85,B 0,C 180,E1 -13528.893,E2 -13528.893} C_VEL
LIN {X 0,Y 475.428,Z 442.959,A -85,B 0,C 180,E1 -13530.633,E2 -13530.633} C_VEL
LIN {X 0,Y 480.616,Z 390.245,A -85,B 0,C 180,E1 -13534.681,E2 -13534.681} C_VEL
LIN {X 0,Y 486.158,Z 339.219,A -85,B 0,C 180,E1 -13538.625,E2 -13538.625} C_VEL
LIN {X 0,Y 489.964,Z 306.282,A -85,B 0,C 180,E1 -13541.19,E2 -13541.19} C_VEL
LIN {X 0,Y 486.224,Z 295.751,A -85,B 0,C 180,E1 -13542.488,E2 -13542.488} C_VEL
LIN {X 0,Y 488.357,Z 296.309,A -85,B 0,C 180,E1 -13542.825,E2 -13542.825} C_VEL
LIN {X 0,Y 494.683,Z 296.459,A -85,B 0,C 180,E1 -13543.691,E2 -13543.691} C_VEL
LIN {X 0,Y 502.56,Z 316.624,A -85,B 0,C 180,E1 -13546.239,E2 -13546.239} C_VEL
LIN {X 0,Y 505.822,Z 326.064,A -85,B 0,C 180,E1 -13547.338,E2 -13547.338} C_VEL
LIN {X 0,Y 505.293,Z 362.094,A -85,B 0,C 180,E1 -13549.827,E2 -13549.827} C_VEL
LIN {X 0,Y 501.139,Z 381.657,A -85,B 0,C 180,E1 -13550.552,E2 -13550.552} C_VEL
LIN {X 0,Y 497.822,Z 466.245,A -85,B 0,C 180,E1 -13551.885,E2 -13551.885} C_VEL
LIN {X 0,Y 494.1,Z 533.338,A -85,B 0,C 180,E1 -13553.138,E2 -13553.138} C_VEL
LIN {X 0,Y 490.025,Z 593.617,A -85,B 0,C 180,E1 -13554.426,E2 -13554.426} C_VEL
LIN {X 0,Y 488.675,Z 601.21,A -85,B 0,C 180,E1 -13554.531,E2 -13554.531} C_VEL
LIN {X 0,Y 482.152,Z 621.424,A -85,B 0,C 180,E1 -13554.569,E2 -13554.569} C_VEL
LIN {X 0,Y 481.085,Z 627.928,A -85,B 0,C 180,E1 -13554.677,E2 -13554.677} C_VEL
LIN {X 0,Y 479.076,Z 661.98,A -85,B 0,C 180,E1 -13555.628,E2 -13555.628} C_VEL
LIN {X 0,Y 477.368,Z 684.08,A -85,B 0,C 180,E1 -13556.476,E2 -13556.476} C_VEL
LIN {X 0,Y 475.188,Z 705.766,A -85,B 0,C 180,E1 -13557.549,E2 -13557.549} C_VEL
LIN {X 0,Y 472.71,Z 725.9,A -85,B 0,C 180,E1 -13558.786,E2 -13558.786} C_VEL
LIN {X 0,Y 469.934,Z 745.461,A -85,B 0,C 180,E1 -13560.241,E2 -13560.241} C_VEL
LIN {X 0,Y 467.104,Z 763.42,A -85,B 0,C 180,E1 -13561.835,E2 -13561.835} C_VEL
LIN {X 0,Y 464.147,Z 780.829,A -85,B 0,C 180,E1 -13563.66,E2 -13563.66} C_VEL
LIN {X 0,Y 461.249,Z 797.096,A -85,B 0,C 180,E1 -13565.677,E2 -13565.677} C_VEL
LIN {X 0,Y 458.555,Z 811.859,A -85,B 0,C 180,E1 -13567.838,E2 -13567.838} C_VEL
LIN {X 0,Y 456.146,Z 825.154,A -85,B 0,C 180,E1 -13570.137,E2 -13570.137} C_VEL
LIN {X 0,Y 454.078,Z 836.979,A -85,B 0,C 180,E1 -13572.574,E2 -13572.574} C_VEL
LIN {X 0,Y 452.378,Z 847.3,A -85,B 0,C 180,E1 -13575.144,E2 -13575.144} C_VEL
LIN {X 0,Y 451.083,Z 856.031,A -85,B 0,C 180,E1 -13577.843,E2 -13577.843} C_VEL
LIN {X 0,Y 450.214,Z 862.595,A -85,B 0,C 180,E1 -13580.434,E2 -13580.434} C_VEL
LIN {X 0,Y 449.668,Z 867.666,A -85,B 0,C 180,E1 -13583.103,E2 -13583.103} C_VEL
LIN {X 0,Y 449.371,Z 871.007,A -85,B 0,C 180,E1 -13585.661,E2 -13585.661} C_VEL
LIN {X 0,Y 449.224,Z 872.865,A -85,B 0,C 180,E1 -13588.342,E2 -13588.342} C_VEL
LIN {X 0,Y 449.198,Z 873.077,A -85,B 0,C 180,E1 -13590.893,E2 -13590.893} C_VEL
LIN {X 0,Y 449.3,Z 871.752,A -85,B 0,C 180,E1 -13593.572,E2 -13593.572} C_VEL
LIN {X 0,Y 449.556,Z 868.955,A -85,B 0,C 180,E1 -13596.168,E2 -13596.168} C_VEL
LIN {X 0,Y 450.042,Z 864.162,A -85,B 0,C 180,E1 -13598.947,E2 -13598.947} C_VEL
LIN {X 0,Y 450.791,Z 858.057,A -85,B 0,C 180,E1 -13601.515,E2 -13601.515} C_VEL
LIN {X 0,Y 451.971,Z 849.84,A -85,B 0,C 180,E1 -13604.215,E2 -13604.215} C_VEL
LIN {X 0,Y 453.537,Z 840.114,A -85,B 0,C 180,E1 -13606.787,E2 -13606.787} C_VEL
LIN {X 0,Y 455.484,Z 828.952,A -85,B 0,C 180,E1 -13609.225,E2 -13609.225} C_VEL
LIN {X 0,Y 457.768,Z 816.401,A -85,B 0,C 180,E1 -13611.528,E2 -13611.528} C_VEL
LIN {X 0,Y 460.491,Z 801.535,A -85,B 0,C 180,E1 -13613.82,E2 -13613.82} C_VEL
LIN {X 0,Y 463.393,Z 785.44,A -85,B 0,C 180,E1 -13615.909,E2 -13615.909} C_VEL
LIN {X 0,Y 466.333,Z 768.344,A -85,B 0,C 180,E1 -13617.784,E2 -13617.784} C_VEL
LIN {X 0,Y 469.068,Z 751.399,A -85,B 0,C 180,E1 -13619.359,E2 -13619.359} C_VEL
LIN {X 0,Y 471.842,Z 732.449,A -85,B 0,C 180,E1 -13620.852,E2 -13620.852} C_VEL
LIN {X 0,Y 474.38,Z 712.797,A -85,B 0,C 180,E1 -13622.142,E2 -13622.142} C_VEL
LIN {X 0,Y 476.62,Z 692.451,A -85,B 0,C 180,E1 -13623.235,E2 -13623.235} C_VEL
LIN {X 0,Y 478.464,Z 671.503,A -85,B 0,C 180,E1 -13624.133,E2 -13624.133} C_VEL
LIN {X 0,Y 479.862,Z 649.328,A -85,B 0,C 180,E1 -13624.856,E2 -13624.856} C_VEL
LIN {X 0,Y 482.942,Z 603.252,A -85,B 0,C 180,E1 -13626.015,E2 -13626.015} C_VEL
LIN {X 0,Y 487.734,Z 535.64,A -85,B 0,C 180,E1 -13627.496,E2 -13627.496} C_VEL
LIN {X 0,Y 491.458,Z 471.348,A -85,B 0,C 180,E1 -13628.716,E2 -13628.716} C_VEL
LIN {X 0,Y 494.698,Z 393.121,A -85,B 0,C 180,E1 -13629.971,E2 -13629.971} C_VEL
LIN {X 0,Y 495.169,Z 382.888,A -85,B 0,C 180,E1 -13630.14,E2 -13630.14} C_VEL
LIN {X 0,Y 499.455,Z 363.438,A -85,B 0,C 180,E1 -13630.892,E2 -13630.892} C_VEL
LIN {X 0,Y 499.819,Z 329.349,A -85,B 0,C 180,E1 -13633.265,E2 -13633.265} C_VEL
LIN {X 0,Y 492.328,Z 309.141,A -85,B 0,C 180,E1 -13635.763,E2 -13635.763} C_VEL
LIN {X 0,Y 484.713,Z 291.025,A -85,B 0,C 180,E1 -13638.218,E2 -13638.218} C_VEL
LIN {X 0,Y 477.071,Z 275.122,A -85,B 0,C 180,E1 -13640.576,E2 -13640.576} C_VEL
LIN {X 0,Y 470.415,Z 262.693,A -85,B 0,C 180,E1 -13642.561,E2 -13642.561} C_VEL
LIN {X 0,Y 464.9,Z 253.177,A -85,B 0,C 180,E1 -13644.196,E2 -13644.196} C_VEL
LIN {X 0,Y 462.135,Z 248.659,A -85,B 0,C 180,E1 -13645.015,E2 -13645.015} C_VEL
LIN {X 0,Y 459.823,Z 244.742,A -85,B 0,C 180,E1 -13645.722,E2 -13645.722} C_VEL
LIN {X 0,Y 457.513,Z 240.985,A -85,B 0,C 180,E1 -13646.432,E2 -13646.432} C_VEL
LIN {X 0,Y 456.303,Z 239.305,A -85,B 0,C 180,E1 -13646.782,E2 -13646.782} C_VEL
LIN {X 0,Y 454.022,Z 235.539,A -85,B 0,C 180,E1 -13647.496,E2 -13647.496} C_VEL
LIN {X 0,Y 453.254,Z 234.387,A -85,B 0,C 180,E1 -13647.733,E2 -13647.733} C_VEL
LIN {X 0,Y 451.199,Z 231.945,A -85,B 0,C 180,E1 -13648.317,E2 -13648.317} C_VEL
LIN {X 0,Y 450.296,Z 229.13,A -85,B 0,C 180,E1 -13648.748,E2 -13648.748} C_VEL
LIN {X 0,Y 450.293,Z 229.11,A -85,B 0,C 180,E1 -13652.492,E2 -13652.492} C_VEL
LIN {X 0,Y 450.286,Z 229.098,A -85,B 0,C 180,E1 -13656.188,E2 -13656.188} C_VEL
LIN {X 0,Y 450.291,Z 229.127,A -85,B 0,C 180,E1 -13659.933,E2 -13659.933} C_VEL
LIN {X 0,Y 450.291,Z 229.116,A -85,B 0,C 180,E1 -13663.62,E2 -13663.62} C_VEL
LIN {X 0,Y 450.288,Z 229.092,A -85,B 0,C 180,E1 -13667.301,E2 -13667.301} C_VEL
LIN {X 0,Y 450.295,Z 229.139,A -85,B 0,C 180,E1 -13671.058,E2 -13671.058} C_VEL
LIN {X 0,Y 450.283,Z 229.094,A -85,B 0,C 180,E1 -13674.776,E2 -13674.776} C_VEL
LIN {X 0,Y 450.278,Z 229.126,A -85,B 0,C 180,E1 -13678.473,E2 -13678.473} C_VEL
LIN {X 0,Y 450.274,Z 229.113,A -85,B 0,C 180,E1 -13682.291,E2 -13682.291} C_VEL
LIN {X 0,Y 450.283,Z 229.099,A -85,B 0,C 180,E1 -13685.991,E2 -13685.991} C_VEL
LIN {X 0,Y 450.294,Z 229.133,A -85,B 0,C 180,E1 -13689.716,E2 -13689.716} C_VEL
LIN {X 0,Y 450.3,Z 229.139,A -85,B 0,C 180,E1 -13693.483,E2 -13693.483} C_VEL
LIN {X 0,Y 450.292,Z 229.142,A -85,B 0,C 180,E1 -13697.177,E2 -13697.177} C_VEL
LIN {X 0,Y 450.271,Z 229.136,A -85,B 0,C 180,E1 -13700.812,E2 -13700.812} C_VEL
LIN {X 0,Y 450.313,Z 229.351,A -85,B 0,C 180,E1 -13704.066,E2 -13704.066} C_VEL
LIN {X 0,Y 451.415,Z 232.38,A -85,B 0,C 180,E1 -13704.609,E2 -13704.609} C_VEL
LIN {X 0,Y 452.816,Z 234.512,A -85,B 0,C 180,E1 -13705.085,E2 -13705.085} C_VEL
LIN {X 0,Y 460.155,Z 248.689,A -85,B 0,C 180,E1 -13707.852,E2 -13707.852} C_VEL
LIN {X 0,Y 468.901,Z 265.678,A -85,B 0,C 180,E1 -13710.925,E2 -13710.925} C_VEL
LIN {X 0,Y 478.993,Z 285.851,A -85,B 0,C 180,E1 -13714.245,E2 -13714.245} C_VEL
LIN {X 0,Y 489.169,Z 306.954,A -85,B 0,C 180,E1 -13717.379,E2 -13717.379} C_VEL
LIN {X 0,Y 496.135,Z 321.396,A -85,B 0,C 180,E1 -13719.333,E2 -13719.333} C_VEL
LIN {X 0,Y 504.323,Z 334.524,A -85,B 0,C 180,E1 -13720.418,E2 -13720.418} C_VEL
LIN {X 0,Y 505.676,Z 351.379,A -85,B 0,C 180,E1 -13720.93,E2 -13720.93} C_VEL
LIN {X 0,Y 493.439,Z 594.424,A -85,B 0,C 180,E1 -13725.177,E2 -13725.177} C_VEL
LIN {X 0,Y 489.052,Z 693.147,A -85,B 0,C 180,E1 -13726.899,E2 -13726.899} C_VEL
LIN {X 0,Y 487.064,Z 717.705,A -85,B 0,C 180,E1 -13727.52,E2 -13727.52} C_VEL
LIN {X 0,Y 484.689,Z 741.475,A -85,B 0,C 180,E1 -13728.313,E2 -13728.313} C_VEL
LIN {X 0,Y 482.008,Z 763.641,A -85,B 0,C 180,E1 -13729.256,E2 -13729.256} C_VEL
LIN {X 0,Y 478.771,Z 787.263,A -85,B 0,C 180,E1 -13730.479,E2 -13730.479} C_VEL
LIN {X 0,Y 475.64,Z 807.713,A -85,B 0,C 180,E1 -13731.75,E2 -13731.75} C_VEL
LIN {X 0,Y 471.802,Z 830.773,A -85,B 0,C 180,E1 -13733.45,E2 -13733.45} C_VEL
LIN {X 0,Y 468.306,Z 850.667,A -85,B 0,C 180,E1 -13735.17,E2 -13735.17} C_VEL
LIN {X 0,Y 464.826,Z 869.705,A -85,B 0,C 180,E1 -13737.096,E2 -13737.096} C_VEL
LIN {X 0,Y 461.569,Z 887.432,A -85,B 0,C 180,E1 -13739.147,E2 -13739.147} C_VEL
LIN {X 0,Y 458.56,Z 903.615,A -85,B 0,C 180,E1 -13741.334,E2 -13741.334} C_VEL
LIN {X 0,Y 455.749,Z 919.662,A -85,B 0,C 180,E1 -13743.809,E2 -13743.809} C_VEL
LIN {X 0,Y 453.421,Z 933.611,A -85,B 0,C 180,E1 -13746.338,E2 -13746.338} C_VEL
LIN {X 0,Y 451.558,Z 946.259,A -85,B 0,C 180,E1 -13748.979,E2 -13748.979} C_VEL
LIN {X 0,Y 450.159,Z 957.389,A -85,B 0,C 180,E1 -13751.749,E2 -13751.749} C_VEL
LIN {X 0,Y 449.189,Z 967.193,A -85,B 0,C 180,E1 -13754.639,E2 -13754.639} C_VEL
LIN {X 0,Y 448.675,Z 974.712,A -85,B 0,C 180,E1 -13757.385,E2 -13757.385} C_VEL
LIN {X 0,Y 448.445,Z 981.014,A -85,B 0,C 180,E1 -13760.244,E2 -13760.244} C_VEL
LIN {X 0,Y 448.43,Z 985.494,A -85,B 0,C 180,E1 -13763.084,E2 -13763.084} C_VEL
LIN {X 0,Y 448.492,Z 988.15,A -85,B 0,C 180,E1 -13765.525,E2 -13765.525} C_VEL
LIN {X 0,Y 448.566,Z 989.821,A -85,B 0,C 180,E1 -13768.34,E2 -13768.34} C_VEL
LIN {X 0,Y 448.582,Z 989.831,A -85,B 0,C 180,E1 -13771.022,E2 -13771.022} C_VEL
LIN {X 0,Y 448.552,Z 988.674,A -85,B 0,C 180,E1 -13773.451,E2 -13773.451} C_VEL
LIN {X 0,Y 448.472,Z 985.962,A -85,B 0,C 180,E1 -13776.272,E2 -13776.272} C_VEL
LIN {X 0,Y 448.462,Z 981.519,A -85,B 0,C 180,E1 -13779.108,E2 -13779.108} C_VEL
LIN {X 0,Y 448.59,Z 976.15,A -85,B 0,C 180,E1 -13781.703,E2 -13781.703} C_VEL
LIN {X 0,Y 449.049,Z 968.252,A -85,B 0,C 180,E1 -13784.705,E2 -13784.705} C_VEL
LIN {X 0,Y 449.779,Z 959.77,A -85,B 0,C 180,E1 -13787.331,E2 -13787.331} C_VEL
LIN {X 0,Y 451.063,Z 948.711,A -85,B 0,C 180,E1 -13790.231,E2 -13790.231} C_VEL
LIN {X 0,Y 452.845,Z 936.106,A -85,B 0,C 180,E1 -13793.006,E2 -13793.006} C_VEL
LIN {X 0,Y 455.38,Z 920.711,A -85,B 0,C 180,E1 -13795.91,E2 -13795.91} C_VEL
LIN {X 0,Y 458.179,Z 905.313,A -85,B 0,C 180,E1 -13798.408,E2 -13798.408} C_VEL
LIN {X 0,Y 461.612,Z 887.583,A -85,B 0,C 180,E1 -13800.888,E2 -13800.888} C_VEL
LIN {X 0,Y 465.255,Z 869.575,A -85,B 0,C 180,E1 -13803.085,E2 -13803.085} C_VEL
LIN {X 0,Y 469.16,Z 850.023,A -85,B 0,C 180,E1 -13805.13,E2 -13805.13} C_VEL
LIN {X 0,Y 473.357,Z 829.218,A -85,B 0,C 180,E1 -13807.016,E2 -13807.016} C_VEL
LIN {X 0,Y 477.469,Z 807.865,A -85,B 0,C 180,E1 -13808.669,E2 -13808.669} C_VEL
LIN {X 0,Y 481.578,Z 785.351,A -85,B 0,C 180,E1 -13810.142,E2 -13810.142} C_VEL
LIN {X 0,Y 485.477,Z 762.75,A -85,B 0,C 180,E1 -13811.387,E2 -13811.387} C_VEL
LIN {X 0,Y 489.041,Z 739.355,A -85,B 0,C 180,E1 -13812.432,E2 -13812.432} C_VEL
LIN {X 0,Y 492.468,Z 713.955,A -85,B 0,C 180,E1 -13813.33,E2 -13813.33} C_VEL
LIN {X 0,Y 495.235,Z 689.22,A -85,B 0,C 180,E1 -13813.991,E2 -13813.991} C_VEL
LIN {X 0,Y 502.415,Z 606.101,A -85,B 0,C 180,E1 -13815.717,E2 -13815.717} C_VEL
LIN {X 0,Y 509.652,Z 543.883,A -85,B 0,C 180,E1 -13817.107,E2 -13817.107} C_VEL
LIN {X 0,Y 518.608,Z 484.008,A -85,B 0,C 180,E1 -13818.523,E2 -13818.523} C_VEL
LIN {X 0,Y 529.824,Z 424.254,A -85,B 0,C 180,E1 -13819.952,E2 -13819.952} C_VEL
LIN {X 0,Y 530.345,Z 421.728,A -85,B 0,C 180,E1 -13820.022,E2 -13820.022} C_VEL
LIN {X 0,Y 525.481,Z 439.424,A -85,B 0,C 180,E1 -13821.347,E2 -13821.347} C_VEL
LIN {X 0,Y 521.194,Z 459.651,A -85,B 0,C 180,E1 -13822.691,E2 -13822.691} C_VEL
LIN {X 0,Y 517.046,Z 484.385,A -85,B 0,C 180,E1 -13824.138,E2 -13824.138} C_VEL
LIN {X 0,Y 512.915,Z 514.472,A -85,B 0,C 180,E1 -13825.684,E2 -13825.684} C_VEL
LIN {X 0,Y 511.601,Z 522.309,A -85,B 0,C 180,E1 -13825.939,E2 -13825.939} C_VEL
LIN {X 0,Y 494.044,Z 627.424,A -85,B 0,C 180,E1 -13828.967,E2 -13828.967} C_VEL
LIN {X 0,Y 484.529,Z 693.436,A -85,B 0,C 180,E1 -13830.974,E2 -13830.974} C_VEL
LIN {X 0,Y 480.673,Z 717.867,A -85,B 0,C 180,E1 -13831.958,E2 -13831.958} C_VEL
LIN {X 0,Y 476.883,Z 740.991,A -85,B 0,C 180,E1 -13833.138,E2 -13833.138} C_VEL
LIN {X 0,Y 473.152,Z 763.244,A -85,B 0,C 180,E1 -13834.529,E2 -13834.529} C_VEL
LIN {X 0,Y 469.661,Z 783.67,A -85,B 0,C 180,E1 -13836.073,E2 -13836.073} C_VEL
LIN {X 0,Y 466.419,Z 802.263,A -85,B 0,C 180,E1 -13837.767,E2 -13837.767} C_VEL
LIN {X 0,Y 463.679,Z 817.604,A -85,B 0,C 180,E1 -13839.421,E2 -13839.421} C_VEL
LIN {X 0,Y 461.038,Z 832.136,A -85,B 0,C 180,E1 -13841.278,E2 -13841.278} C_VEL
LIN {X 0,Y 458.61,Z 845.081,A -85,B 0,C 180,E1 -13843.274,E2 -13843.274} C_VEL
LIN {X 0,Y 456.552,Z 855.769,A -85,B 0,C 180,E1 -13845.283,E2 -13845.283} C_VEL
LIN {X 0,Y 454.829,Z 864.486,A -85,B 0,C 180,E1 -13847.3,E2 -13847.3} C_VEL
LIN {X 0,Y 453.255,Z 872.152,A -85,B 0,C 180,E1 -13849.578,E2 -13849.578} C_VEL
LIN {X 0,Y 452.041,Z 877.742,A -85,B 0,C 180,E1 -13851.862,E2 -13851.862} C_VEL
LIN {X 0,Y 451.139,Z 881.424,A -85,B 0,C 180,E1 -13854.148,E2 -13854.148} C_VEL
LIN {X 0,Y 450.515,Z 883.217,A -85,B 0,C 180,E1 -13856.31,E2 -13856.31} C_VEL
LIN {X 0,Y 450.074,Z 883.39,A -85,B 0,C 180,E1 -13858.6,E2 -13858.6} C_VEL
LIN {X 0,Y 449.815,Z 881.823,A -85,B 0,C 180,E1 -13860.892,E2 -13860.892} C_VEL
LIN {X 0,Y 449.716,Z 878.498,A -85,B 0,C 180,E1 -13863.186,E2 -13863.186} C_VEL
LIN {X 0,Y 449.795,Z 873.387,A -85,B 0,C 180,E1 -13865.485,E2 -13865.485} C_VEL
LIN {X 0,Y 450.067,Z 866.52,A -85,B 0,C 180,E1 -13867.753,E2 -13867.753} C_VEL
LIN {X 0,Y 450.558,Z 857.917,A -85,B 0,C 180,E1 -13869.968,E2 -13869.968} C_VEL
LIN {X 0,Y 451.318,Z 847.405,A -85,B 0,C 180,E1 -13872.15,E2 -13872.15} C_VEL
LIN {X 0,Y 452.311,Z 835.396,A -85,B 0,C 180,E1 -13874.204,E2 -13874.204} C_VEL
LIN {X 0,Y 453.613,Z 820.956,A -85,B 0,C 180,E1 -13876.257,E2 -13876.257} C_VEL
LIN {X 0,Y 455.089,Z 805.309,A -85,B 0,C 180,E1 -13878.113,E2 -13878.113} C_VEL
LIN {X 0,Y 456.753,Z 787.953,A -85,B 0,C 180,E1 -13879.835,E2 -13879.835} C_VEL
LIN {X 0,Y 458.462,Z 769.351,A -85,B 0,C 180,E1 -13881.365,E2 -13881.365} C_VEL
LIN {X 0,Y 460.196,Z 749.84,A -85,B 0,C 180,E1 -13882.685,E2 -13882.685} C_VEL
LIN {X 0,Y 461.88,Z 729.249,A -85,B 0,C 180,E1 -13883.812,E2 -13883.812} C_VEL
LIN {X 0,Y 463.467,Z 707.122,A -85,B 0,C 180,E1 -13884.76,E2 -13884.76} C_VEL
LIN {X 0,Y 464.819,Z 685.119,A -85,B 0,C 180,E1 -13885.452,E2 -13885.452} C_VEL
LIN {X 0,Y 473.257,Z 502.713,A -85,B 0,C 180,E1 -13889.308,E2 -13889.308} C_VEL
LIN {X 0,Y 468.265,Z 442.042,A -85,B 0,C 180,E1 -13891.15,E2 -13891.15} C_VEL
LIN {X 0,Y 473.624,Z 389.762,A -85,B 0,C 180,E1 -13895.213,E2 -13895.213} C_VEL
LIN {X 0,Y 479.379,Z 338.841,A -85,B 0,C 180,E1 -13899.198,E2 -13899.198} C_VEL
LIN {X 0,Y 482.929,Z 309.227,A -85,B 0,C 180,E1 -13901.532,E2 -13901.532} C_VEL
LIN {X 0,Y 480.743,Z 303.161,A -85,B 0,C 180,E1 -13902.287,E2 -13902.287} C_VEL
LIN {X 0,Y 482.802,Z 303.744,A -85,B 0,C 180,E1 -13902.627,E2 -13902.627} C_VEL
LIN {X 0,Y 490.134,Z 303.685,A -85,B 0,C 180,E1 -13903.634,E2 -13903.634} C_VEL
LIN {X 0,Y 497.91,Z 324.114,A -85,B 0,C 180,E1 -13906.215,E2 -13906.215} C_VEL
LIN {X 0,Y 499.866,Z 330.008,A -85,B 0,C 180,E1 -13906.896,E2 -13906.896} C_VEL
LIN {X 0,Y 499.283,Z 364.047,A -85,B 0,C 180,E1 -13909.242,E2 -13909.242} C_VEL
LIN {X 0,Y 494.952,Z 384.388,A -85,B 0,C 180,E1 -13909.995,E2 -13909.995} C_VEL
LIN {X 0,Y 491.542,Z 468.475,A -85,B 0,C 180,E1 -13911.331,E2 -13911.331} C_VEL
LIN {X 0,Y 487.771,Z 534.231,A -85,B 0,C 180,E1 -13912.574,E2 -13912.574} C_VEL
LIN {X 0,Y 482.681,Z 606.165,A -85,B 0,C 180,E1 -13914.15,E2 -13914.15} C_VEL
LIN {X 0,Y 481.085,Z 627.928,A -85,B 0,C 180,E1 -13914.677,E2 -13914.677} C_VEL
LIN {X 0,Y 479.763,Z 635.517,A -85,B 0,C 180,E1 -13914.8,E2 -13914.8} C_VEL
LIN {X 0,Y 473.715,Z 654.685,A -85,B 0,C 180,E1 -13914.902,E2 -13914.902} C_VEL
LIN {X 0,Y 472.525,Z 662.213,A -85,B 0,C 180,E1 -13915.072,E2 -13915.072} C_VEL
LIN {X 0,Y 470.817,Z 683.781,A -85,B 0,C 180,E1 -13915.898,E2 -13915.898} C_VEL
LIN {X 0,Y 468.734,Z 704.222,A -85,B 0,C 180,E1 -13916.901,E2 -13916.901} C_VEL
LIN {X 0,Y 466.184,Z 724.726,A -85,B 0,C 180,E1 -13918.142,E2 -13918.142} C_VEL
LIN {X 0,Y 463.318,Z 744.487,A -85,B 0,C 180,E1 -13919.599,E2 -13919.599} C_VEL
LIN {X 0,Y 460.204,Z 763.725,A -85,B 0,C 180,E1 -13921.303,E2 -13921.303} C_VEL
LIN {X 0,Y 457.019,Z 781.761,A -85,B 0,C 180,E1 -13923.211,E2 -13923.211} C_VEL
LIN {X 0,Y 453.984,Z 798.079,A -85,B 0,C 180,E1 -13925.262,E2 -13925.262} C_VEL
LIN {X 0,Y 451.166,Z 812.861,A -85,B 0,C 180,E1 -13927.455,E2 -13927.455} C_VEL
LIN {X 0,Y 448.637,Z 826.157,A -85,B 0,C 180,E1 -13929.79,E2 -13929.79} C_VEL
LIN {X 0,Y 446.458,Z 837.988,A -85,B 0,C 180,E1 -13932.267,E2 -13932.267} C_VEL
LIN {X 0,Y 444.658,Z 848.297,A -85,B 0,C 180,E1 -13934.88,E2 -13934.88} C_VEL
LIN {X 0,Y 443.284,Z 857.031,A -85,B 0,C 180,E1 -13937.626,E2 -13937.626} C_VEL
LIN {X 0,Y 442.358,Z 863.547,A -85,B 0,C 180,E1 -13940.24,E2 -13940.24} C_VEL
LIN {X 0,Y 441.767,Z 868.671,A -85,B 0,C 180,E1 -13942.979,E2 -13942.979} C_VEL
LIN {X 0,Y 441.434,Z 872.12,A -85,B 0,C 180,E1 -13945.713,E2 -13945.713} C_VEL
LIN {X 0,Y 441.285,Z 873.933,A -85,B 0,C 180,E1 -13948.442,E2 -13948.442} C_VEL
LIN {X 0,Y 441.265,Z 874.056,A -85,B 0,C 180,E1 -13951.039,E2 -13951.039} C_VEL
LIN {X 0,Y 441.381,Z 872.641,A -85,B 0,C 180,E1 -13953.767,E2 -13953.767} C_VEL
LIN {X 0,Y 441.658,Z 869.817,A -85,B 0,C 180,E1 -13956.369,E2 -13956.369} C_VEL
LIN {X 0,Y 442.172,Z 865.168,A -85,B 0,C 180,E1 -13959.108,E2 -13959.108} C_VEL
LIN {X 0,Y 442.974,Z 859.061,A -85,B 0,C 180,E1 -13961.721,E2 -13961.721} C_VEL
LIN {X 0,Y 444.159,Z 851.277,A -85,B 0,C 180,E1 -13964.337,E2 -13964.337} C_VEL
LIN {X 0,Y 445.794,Z 841.651,A -85,B 0,C 180,E1 -13966.953,E2 -13966.953} C_VEL
LIN {X 0,Y 447.823,Z 830.601,A -85,B 0,C 180,E1 -13969.432,E2 -13969.432} C_VEL
LIN {X 0,Y 450.273,Z 817.754,A -85,B 0,C 180,E1 -13971.84,E2 -13971.84} C_VEL
LIN {X 0,Y 453.021,Z 803.399,A -85,B 0,C 180,E1 -13974.1,E2 -13974.1} C_VEL
LIN {X 0,Y 456.029,Z 787.439,A -85,B 0,C 180,E1 -13976.219,E2 -13976.219} C_VEL
LIN {X 0,Y 459.015,Z 770.826,A -85,B 0,C 180,E1 -13978.087,E2 -13978.087} C_VEL
LIN {X 0,Y 461.904,Z 753.768,A -85,B 0,C 180,E1 -13979.717,E2 -13979.717} C_VEL
LIN {X 0,Y 464.9,Z 734.209,A -85,B 0,C 180,E1 -13981.293,E2 -13981.293} C_VEL
LIN {X 0,Y 467.548,Z 714.477,A -85,B 0,C 180,E1 -13982.61,E2 -13982.61} C_VEL
LIN {X 0,Y 469.84,Z 694.497,A -85,B 0,C 180,E1 -13983.704,E2 -13983.704} C_VEL
LIN {X 0,Y 471.765,Z 673.569,A -85,B 0,C 180,E1 -13984.621,E2 -13984.621} C_VEL
LIN {X 0,Y 473.232,Z 651.389,A -85,B 0,C 180,E1 -13985.362,E2 -13985.362} C_VEL
LIN {X 0,Y 476.293,Z 606.899,A -85,B 0,C 180,E1 -13986.51,E2 -13986.51} C_VEL
LIN {X 0,Y 481.206,Z 540.255,A -85,B 0,C 180,E1 -13987.998,E2 -13987.998} C_VEL
LIN {X 0,Y 485.108,Z 475.854,A -85,B 0,C 180,E1 -13989.244,E2 -13989.244} C_VEL
LIN {X 0,Y 488.427,Z 399.113,A -85,B 0,C 180,E1 -13990.491,E2 -13990.491} C_VEL
LIN {X 0,Y 489.027,Z 385.666,A -85,B 0,C 180,E1 -13990.711,E2 -13990.711} C_VEL
LIN {X 0,Y 493.565,Z 365.343,A -85,B 0,C 180,E1 -13991.487,E2 -13991.487} C_VEL
LIN {X 0,Y 493.921,Z 333.3,A -85,B 0,C 180,E1 -13993.721,E2 -13993.721} C_VEL
LIN {X 0,Y 486.305,Z 312.723,A -85,B 0,C 180,E1 -13996.302,E2 -13996.302} C_VEL
LIN {X 0,Y 478.6,Z 294.408,A -85,B 0,C 180,E1 -13998.845,E2 -13998.845} C_VEL
LIN {X 0,Y 470.59,Z 277.843,A -85,B 0,C 180,E1 -14001.341,E2 -14001.341} C_VEL
LIN {X 0,Y 463.675,Z 264.985,A -85,B 0,C 180,E1 -14003.474,E2 -14003.474} C_VEL
LIN {X 0,Y 457.471,Z 254.543,A -85,B 0,C 180,E1 -14005.369,E2 -14005.369} C_VEL
LIN {X 0,Y 455.192,Z 250.74,A -85,B 0,C 180,E1 -14006.086,E2 -14006.086} C_VEL
LIN {X 0,Y 452.103,Z 245.816,A -85,B 0,C 180,E1 -14007.039,E2 -14007.039} C_VEL
LIN {X 0,Y 449.837,Z 242.202,A -85,B 0,C 180,E1 -14007.76,E2 -14007.76} C_VEL
LIN {X 0,Y 448.675,Z 240.567,A -85,B 0,C 180,E1 -14008.118,E2 -14008.118} C_VEL
LIN {X 0,Y 446.433,Z 237.103,A -85,B 0,C 180,E1 -14008.843,E2 -14008.843} C_VEL
LIN {X 0,Y 445.754,Z 235.733,A -85,B 0,C 180,E1 -14009.091,E2 -14009.091} C_VEL
LIN {X 0,Y 443.354,Z 233.096,A -85,B 0,C 180,E1 -14009.806,E2 -14009.806} C_VEL
LIN {X 0,Y 442.354,Z 230.106,A -85,B 0,C 180,E1 -14010.289,E2 -14010.289} C_VEL
LIN {X 0,Y 442.354,Z 230.128,A -85,B 0,C 180,E1 -14014.135,E2 -14014.135} C_VEL
LIN {X 0,Y 442.354,Z 230.101,A -85,B 0,C 180,E1 -14017.962,E2 -14017.962} C_VEL
LIN {X 0,Y 442.351,Z 230.08,A -85,B 0,C 180,E1 -14021.689,E2 -14021.689} C_VEL
LIN {X 0,Y 442.353,Z 230.117,A -85,B 0,C 180,E1 -14025.469,E2 -14025.469} C_VEL
LIN {X 0,Y 442.351,Z 230.097,A -85,B 0,C 180,E1 -14029.318,E2 -14029.318} C_VEL
LIN {X 0,Y 442.357,Z 230.083,A -85,B 0,C 180,E1 -14033.119,E2 -14033.119} C_VEL
LIN {X 0,Y 442.349,Z 230.128,A -85,B 0,C 180,E1 -14036.89,E2 -14036.89} C_VEL
LIN {X 0,Y 442.337,Z 230.076,A -85,B 0,C 180,E1 -14040.648,E2 -14040.648} C_VEL
LIN {X 0,Y 442.336,Z 230.128,A -85,B 0,C 180,E1 -14044.408,E2 -14044.408} C_VEL
LIN {X 0,Y 442.334,Z 230.084,A -85,B 0,C 180,E1 -14048.187,E2 -14048.187} C_VEL
LIN {X 0,Y 442.352,Z 230.13,A -85,B 0,C 180,E1 -14051.87,E2 -14051.87} C_VEL
LIN {X 0,Y 442.361,Z 230.116,A -85,B 0,C 180,E1 -14055.654,E2 -14055.654} C_VEL
LIN {X 0,Y 442.36,Z 230.122,A -85,B 0,C 180,E1 -14059.407,E2 -14059.407} C_VEL
LIN {X 0,Y 442.336,Z 230.175,A -85,B 0,C 180,E1 -14062.81,E2 -14062.81} C_VEL
LIN {X 0,Y 443.713,Z 233.671,A -85,B 0,C 180,E1 -14063.486,E2 -14063.486} C_VEL
LIN {X 0,Y 444.82,Z 235.229,A -85,B 0,C 180,E1 -14063.867,E2 -14063.867} C_VEL
LIN {X 0,Y 446.588,Z 238.926,A -85,B 0,C 180,E1 -14064.611,E2 -14064.611} C_VEL
LIN {X 0,Y 452.364,Z 249.899,A -85,B 0,C 180,E1 -14066.803,E2 -14066.803} C_VEL
LIN {X 0,Y 459.607,Z 263.997,A -85,B 0,C 180,E1 -14069.451,E2 -14069.451} C_VEL
LIN {X 0,Y 469.317,Z 283.159,A -85,B 0,C 180,E1 -14072.762,E2 -14072.762} C_VEL
LIN {X 0,Y 479.486,Z 304.083,A -85,B 0,C 180,E1 -14076.02,E2 -14076.02} C_VEL
LIN {X 0,Y 488.185,Z 322.254,A -85,B 0,C 180,E1 -14078.566,E2 -14078.566} C_VEL
LIN {X 0,Y 498.33,Z 338.535,A -85,B 0,C 180,E1 -14079.947,E2 -14079.947} C_VEL
LIN {X 0,Y 499.433,Z 352.494,A -85,B 0,C 180,E1 -14080.368,E2 -14080.368} C_VEL
LIN {X 0,Y 486.734,Z 594.185,A -85,B 0,C 180,E1 -14084.663,E2 -14084.663} C_VEL
LIN {X 0,Y 482.147,Z 693.173,A -85,B 0,C 180,E1 -14086.421,E2 -14086.421} C_VEL
LIN {X 0,Y 480.107,Z 717.55,A -85,B 0,C 180,E1 -14087.049,E2 -14087.049} C_VEL
LIN {X 0,Y 477.638,Z 741.517,A -85,B 0,C 180,E1 -14087.861,E2 -14087.861} C_VEL
LIN {X 0,Y 474.804,Z 764.239,A -85,B 0,C 180,E1 -14088.845,E2 -14088.845} C_VEL
LIN {X 0,Y 471.297,Z 788.852,A -85,B 0,C 180,E1 -14090.155,E2 -14090.155} C_VEL
LIN {X 0,Y 468.02,Z 809.633,A -85,B 0,C 180,E1 -14091.481,E2 -14091.481} C_VEL
LIN {X 0,Y 464.382,Z 830.763,A -85,B 0,C 180,E1 -14093.078,E2 -14093.078} C_VEL
LIN {X 0,Y 460.669,Z 851.372,A -85,B 0,C 180,E1 -14094.887,E2 -14094.887} C_VEL
LIN {X 0,Y 457.099,Z 870.27,A -85,B 0,C 180,E1 -14096.848,E2 -14096.848} C_VEL
LIN {X 0,Y 453.612,Z 888.611,A -85,B 0,C 180,E1 -14099.034,E2 -14099.034} C_VEL
LIN {X 0,Y 450.609,Z 904.415,A -85,B 0,C 180,E1 -14101.223,E2 -14101.223} C_VEL
LIN {X 0,Y 447.737,Z 920.352,A -85,B 0,C 180,E1 -14103.757,E2 -14103.757} C_VEL
LIN {X 0,Y 445.513,Z 933.366,A -85,B 0,C 180,E1 -14106.173,E2 -14106.173} C_VEL
LIN {X 0,Y 443.525,Z 946.498,A -85,B 0,C 180,E1 -14108.995,E2 -14108.995} C_VEL
LIN {X 0,Y 442.234,Z 956.556,A -85,B 0,C 180,E1 -14111.546,E2 -14111.546} C_VEL
LIN {X 0,Y 441.234,Z 966.379,A -85,B 0,C 180,E1 -14114.49,E2 -14114.49} C_VEL
LIN {X 0,Y 440.71,Z 973.894,A -85,B 0,C 180,E1 -14117.287,E2 -14117.287} C_VEL
LIN {X 0,Y 440.479,Z 980.191,A -85,B 0,C 180,E1 -14120.198,E2 -14120.198} C_VEL
LIN {X 0,Y 440.472,Z 984.655,A -85,B 0,C 180,E1 -14123.09,E2 -14123.09} C_VEL
LIN {X 0,Y 440.544,Z 987.29,A -85,B 0,C 180,E1 -14125.574,E2 -14125.574} C_VEL
LIN {X 0,Y 440.622,Z 988.907,A -85,B 0,C 180,E1 -14128.44,E2 -14128.44} C_VEL
LIN {X 0,Y 440.64,Z 988.873,A -85,B 0,C 180,E1 -14131.17,E2 -14131.17} C_VEL
LIN {X 0,Y 440.591,Z 987.574,A -85,B 0,C 180,E1 -14133.774,E2 -14133.774} C_VEL
LIN {X 0,Y 440.504,Z 984.504,A -85,B 0,C 180,E1 -14136.779,E2 -14136.779} C_VEL
LIN {X 0,Y 440.507,Z 980.114,A -85,B 0,C 180,E1 -14139.538,E2 -14139.538} C_VEL
LIN {X 0,Y 440.672,Z 974.32,A -85,B 0,C 180,E1 -14142.315,E2 -14142.315} C_VEL
LIN {X 0,Y 441.199,Z 966.109,A -85,B 0,C 180,E1 -14145.376,E2 -14145.376} C_VEL
LIN {X 0,Y 442.052,Z 957.443,A -85,B 0,C 180,E1 -14148.052,E2 -14148.052} C_VEL
LIN {X 0,Y 443.569,Z 945.475,A -85,B 0,C 180,E1 -14151.142,E2 -14151.142} C_VEL
LIN {X 0,Y 445.464,Z 933.249,A -85,B 0,C 180,E1 -14153.83,E2 -14153.83} C_VEL
LIN {X 0,Y 448.123,Z 918.275,A -85,B 0,C 180,E1 -14156.647,E2 -14156.647} C_VEL
LIN {X 0,Y 451.347,Z 901.888,A -85,B 0,C 180,E1 -14159.314,E2 -14159.314} C_VEL
LIN {X 0,Y 454.861,Z 884.689,A -85,B 0,C 180,E1 -14161.71,E2 -14161.71} C_VEL
LIN {X 0,Y 458.989,Z 865.406,A -85,B 0,C 180,E1 -14164.047,E2 -14164.047} C_VEL
LIN {X 0,Y 463.108,Z 846.356,A -85,B 0,C 180,E1 -14166.035,E2 -14166.035} C_VEL
LIN {X 0,Y 467.571,Z 825.15,A -85,B 0,C 180,E1 -14167.938,E2 -14167.938} C_VEL
LIN {X 0,Y 472.033,Z 803.403,A -85,B 0,C 180,E1 -14169.613,E2 -14169.613} C_VEL
LIN {X 0,Y 476.407,Z 780.8,A -85,B 0,C 180,E1 -14171.066,E2 -14171.066} C_VEL
LIN {X 0,Y 480.762,Z 756.468,A -85,B 0,C 180,E1 -14172.366,E2 -14172.366} C_VEL
LIN {X 0,Y 484.653,Z 732.586,A -85,B 0,C 180,E1 -14173.4,E2 -14173.4} C_VEL
LIN {X 0,Y 487.681,Z 710.897,A -85,B 0,C 180,E1 -14174.142,E2 -14174.142} C_VEL
LIN {X 0,Y 490.649,Z 685.393,A -85,B 0,C 180,E1 -14174.813,E2 -14174.813} C_VEL
LIN {X 0,Y 498.083,Z 609.195,A -85,B 0,C 180,E1 -14176.449,E2 -14176.449} C_VEL
LIN {X 0,Y 505.934,Z 548.706,A -85,B 0,C 180,E1 -14177.838,E2 -14177.838} C_VEL
LIN {X 0,Y 515.553,Z 490.353,A -85,B 0,C 180,E1 -14179.242,E2 -14179.242} C_VEL
LIN {X 0,Y 525.388,Z 441.268,A -85,B 0,C 180,E1 -14180.443,E2 -14180.443} C_VEL
LIN {X 0,Y 520.306,Z 461.147,A -85,B 0,C 180,E1 -14181.782,E2 -14181.782} C_VEL
LIN {X 0,Y 515.375,Z 485.401,A -85,B 0,C 180,E1 -14183.235,E2 -14183.235} C_VEL
LIN {X 0,Y 510.589,Z 514.281,A -85,B 0,C 180,E1 -14184.757,E2 -14184.757} C_VEL
LIN {X 0,Y 509.603,Z 520.313,A -85,B 0,C 180,E1 -14185.011,E2 -14185.011} C_VEL
LIN {X 0,Y 490.6,Z 625.827,A -85,B 0,C 180,E1 -14188.082,E2 -14188.082} C_VEL
LIN {X 0,Y 479.982,Z 693.641,A -85,B 0,C 180,E1 -14190.183,E2 -14190.183} C_VEL
LIN {X 0,Y 475.83,Z 717.695,A -85,B 0,C 180,E1 -14191.167,E2 -14191.167} C_VEL
LIN {X 0,Y 471.557,Z 741.406,A -85,B 0,C 180,E1 -14192.399,E2 -14192.399} C_VEL
LIN {X 0,Y 467.523,Z 763.24,A -85,B 0,C 180,E1 -14193.791,E2 -14193.791} C_VEL
LIN {X 0,Y 463.727,Z 783.446,A -85,B 0,C 180,E1 -14195.34,E2 -14195.34} C_VEL
LIN {X 0,Y 460.107,Z 802.686,A -85,B 0,C 180,E1 -14197.108,E2 -14197.108} C_VEL
LIN {X 0,Y 456.73,Z 820.031,A -85,B 0,C 180,E1 -14199.026,E2 -14199.026} C_VEL
LIN {X 0,Y 453.819,Z 834.644,A -85,B 0,C 180,E1 -14200.969,E2 -14200.969} C_VEL
LIN {X 0,Y 451.393,Z 846.564,A -85,B 0,C 180,E1 -14202.866,E2 -14202.866} C_VEL
LIN {X 0,Y 449.196,Z 857.195,A -85,B 0,C 180,E1 -14204.904,E2 -14204.904} C_VEL
LIN {X 0,Y 447.195,Z 866.471,A -85,B 0,C 180,E1 -14207.126,E2 -14207.126} C_VEL
LIN {X 0,Y 445.638,Z 873.434,A -85,B 0,C 180,E1 -14209.267,E2 -14209.267} C_VEL
LIN {X 0,Y 444.323,Z 878.997,A -85,B 0,C 180,E1 -14211.589,E2 -14211.589} C_VEL
LIN {X 0,Y 443.386,Z 882.462,A -85,B 0,C 180,E1 -14213.786,E2 -14213.786} C_VEL
LIN {X 0,Y 442.657,Z 884.395,A -85,B 0,C 180,E1 -14216.114,E2 -14216.114} C_VEL
LIN {X 0,Y 442.173,Z 884.551,A -85,B 0,C 180,E1 -14218.445,E2 -14218.445} C_VEL
LIN {X 0,Y 441.888,Z 882.931,A -85,B 0,C 180,E1 -14220.778,E2 -14220.778} C_VEL
LIN {X 0,Y 441.77,Z 879.587,A -85,B 0,C 180,E1 -14223.114,E2 -14223.114} C_VEL
LIN {X 0,Y 441.842,Z 874.438,A -85,B 0,C 180,E1 -14225.454,E2 -14225.454} C_VEL
LIN {X 0,Y 442.121,Z 867.4,A -85,B 0,C 180,E1 -14227.799,E2 -14227.799} C_VEL
LIN {X 0,Y 442.654,Z 858.321,A -85,B 0,C 180,E1 -14230.148,E2 -14230.148} C_VEL
LIN {X 0,Y 443.451,Z 847.643,A -85,B 0,C 180,E1 -14232.369,E2 -14232.369} C_VEL
LIN {X 0,Y 444.491,Z 835.454,A -85,B 0,C 180,E1 -14234.46,E2 -14234.46} C_VEL
LIN {X 0,Y 445.803,Z 821.309,A -85,B 0,C 180,E1 -14236.483,E2 -14236.483} C_VEL
LIN {X 0,Y 447.334,Z 805.541,A -85,B 0,C 180,E1 -14238.371,E2 -14238.371} C_VEL
LIN {X 0,Y 449.056,Z 788.052,A -85,B 0,C 180,E1 -14240.122,E2 -14240.122} C_VEL
LIN {X 0,Y 450.81,Z 769.422,A -85,B 0,C 180,E1 -14241.668,E2 -14241.668} C_VEL
LIN {X 0,Y 452.615,Z 749.647,A -85,B 0,C 180,E1 -14243.018,E2 -14243.018} C_VEL
LIN {X 0,Y 454.354,Z 728.912,A -85,B 0,C 180,E1 -14244.163,E2 -14244.163} C_VEL
LIN {X 0,Y 455.969,Z 706.942,A -85,B 0,C 180,E1 -14245.112,E2 -14245.112} C_VEL
LIN {X 0,Y 457.382,Z 684.74,A -85,B 0,C 180,E1 -14245.823,E2 -14245.823} C_VEL
LIN {X 0,Y 466.117,Z 503.546,A -85,B 0,C 180,E1 -14249.744,E2 -14249.744} C_VEL
LIN {X 0,Y 461.086,Z 441.386,A -85,B 0,C 180,E1 -14251.654,E2 -14251.654} C_VEL
LIN {X 0,Y 466.557,Z 390.221,A -85,B 0,C 180,E1 -14255.684,E2 -14255.684} C_VEL
LIN {X 0,Y 472.538,Z 339.274,A -85,B 0,C 180,E1 -14259.72,E2 -14259.72} C_VEL
LIN {X 0,Y 475.943,Z 312.332,A -85,B 0,C 180,E1 -14261.862,E2 -14261.862} C_VEL
LIN {X 0,Y 475.392,Z 310.639,A -85,B 0,C 180,E1 -14262.1,E2 -14262.1} C_VEL
LIN {X 0,Y 477.295,Z 311.19,A -85,B 0,C 180,E1 -14262.42,E2 -14262.42} C_VEL
LIN {X 0,Y 485.567,Z 311.009,A -85,B 0,C 180,E1 -14263.577,E2 -14263.577} C_VEL
LIN {X 0,Y 492.952,Z 330.765,A -85,B 0,C 180,E1 -14266.076,E2 -14266.076} C_VEL
LIN {X 0,Y 493.948,Z 333.956,A -85,B 0,C 180,E1 -14266.444,E2 -14266.444} C_VEL
LIN {X 0,Y 493.329,Z 366.026,A -85,B 0,C 180,E1 -14268.643,E2 -14268.643} C_VEL
LIN {X 0,Y 488.809,Z 387.194,A -85,B 0,C 180,E1 -14269.424,E2 -14269.424} C_VEL
LIN {X 0,Y 485.308,Z 470.715,A -85,B 0,C 180,E1 -14270.764,E2 -14270.764} C_VEL
LIN {X 0,Y 481.459,Z 535.724,A -85,B 0,C 180,E1 -14272.006,E2 -14272.006} C_VEL
LIN {X 0,Y 476.291,Z 606.322,A -85,B 0,C 180,E1 -14273.574,E2 -14273.574} C_VEL
LIN {X 0,Y 473.186,Z 651.162,A -85,B 0,C 180,E1 -14274.732,E2 -14274.732} C_VEL
LIN {X 0,Y 472.525,Z 662.213,A -85,B 0,C 180,E1 -14275.072,E2 -14275.072} C_VEL
LIN {X 0,Y 471.236,Z 669.722,A -85,B 0,C 180,E1 -14275.255,E2 -14275.255} C_VEL
LIN {X 0,Y 464.678,Z 688.61,A -85,B 0,C 180,E1 -14275.602,E2 -14275.602} C_VEL
LIN {X 0,Y 463.124,Z 695.785,A -85,B 0,C 180,E1 -14275.876,E2 -14275.876} C_VEL
LIN {X 0,Y 460.73,Z 715.936,A -85,B 0,C 180,E1 -14276.994,E2 -14276.994} C_VEL
LIN {X 0,Y 457.992,Z 735.607,A -85,B 0,C 180,E1 -14278.328,E2 -14278.328} C_VEL
LIN {X 0,Y 454.888,Z 755.12,A -85,B 0,C 180,E1 -14279.923,E2 -14279.923} C_VEL
LIN {X 0,Y 451.639,Z 773.492,A -85,B 0,C 180,E1 -14281.72,E2 -14281.72} C_VEL
LIN {X 0,Y 448.465,Z 790.333,A -85,B 0,C 180,E1 -14283.676,E2 -14283.676} C_VEL
LIN {X 0,Y 445.483,Z 805.483,A -85,B 0,C 180,E1 -14285.748,E2 -14285.748} C_VEL
LIN {X 0,Y 442.719,Z 819.344,A -85,B 0,C 180,E1 -14287.981,E2 -14287.981} C_VEL
LIN {X 0,Y 440.066,Z 832.716,A -85,B 0,C 180,E1 -14290.552,E2 -14290.552} C_VEL
LIN {X 0,Y 437.836,Z 844.411,A -85,B 0,C 180,E1 -14293.277,E2 -14293.277} C_VEL
LIN {X 0,Y 436.113,Z 854.137,A -85,B 0,C 180,E1 -14296.07,E2 -14296.07} C_VEL
LIN {X 0,Y 434.937,Z 861.5,A -85,B 0,C 180,E1 -14298.731,E2 -14298.731} C_VEL
LIN {X 0,Y 434.124,Z 867.452,A -85,B 0,C 180,E1 -14301.523,E2 -14301.523} C_VEL
LIN {X 0,Y 433.632,Z 871.835,A -85,B 0,C 180,E1 -14304.442,E2 -14304.442} C_VEL
LIN {X 0,Y 433.405,Z 874.272,A -85,B 0,C 180,E1 -14307.091,E2 -14307.091} C_VEL
LIN {X 0,Y 433.334,Z 875.196,A -85,B 0,C 180,E1 -14309.868,E2 -14309.868} C_VEL
LIN {X 0,Y 433.377,Z 874.509,A -85,B 0,C 180,E1 -14312.529,E2 -14312.529} C_VEL
LIN {X 0,Y 433.61,Z 872.101,A -85,B 0,C 180,E1 -14315.425,E2 -14315.425} C_VEL
LIN {X 0,Y 434.02,Z 868.367,A -85,B 0,C 180,E1 -14318.078,E2 -14318.078} C_VEL
LIN {X 0,Y 434.792,Z 862.689,A -85,B 0,C 180,E1 -14320.894,E2 -14320.894} C_VEL
LIN {X 0,Y 435.932,Z 855.237,A -85,B 0,C 180,E1 -14323.665,E2 -14323.665} C_VEL
LIN {X 0,Y 437.492,Z 846.246,A -85,B 0,C 180,E1 -14326.327,E2 -14326.327} C_VEL
LIN {X 0,Y 439.441,Z 835.877,A -85,B 0,C 180,E1 -14328.851,E2 -14328.851} C_VEL
LIN {X 0,Y 441.886,Z 823.475,A -85,B 0,C 180,E1 -14331.365,E2 -14331.365} C_VEL
LIN {X 0,Y 444.532,Z 810.383,A -85,B 0,C 180,E1 -14333.602,E2 -14333.602} C_VEL
LIN {X 0,Y 447.552,Z 795.239,A -85,B 0,C 180,E1 -14335.795,E2 -14335.795} C_VEL
LIN {X 0,Y 450.668,Z 779.131,A -85,B 0,C 180,E1 -14337.77,E2 -14337.77} C_VEL
LIN {X 0,Y 453.876,Z 761.355,A -85,B 0,C 180,E1 -14339.61,E2 -14339.61} C_VEL
LIN {X 0,Y 456.985,Z 742.634,A -85,B 0,C 180,E1 -14341.236,E2 -14341.236} C_VEL
LIN {X 0,Y 459.805,Z 723.341,A -85,B 0,C 180,E1 -14342.636,E2 -14342.636} C_VEL
LIN {X 0,Y 462.308,Z 703.547,A -85,B 0,C 180,E1 -14343.82,E2 -14343.82} C_VEL
LIN {X 0,Y 464.501,Z 682.09,A -85,B 0,C 180,E1 -14344.856,E2 -14344.856} C_VEL
LIN {X 0,Y 466.234,Z 659.826,A -85,B 0,C 180,E1 -14345.681,E2 -14345.681} C_VEL
LIN {X 0,Y 469.071,Z 618.252,A -85,B 0,C 180,E1 -14346.831,E2 -14346.831} C_VEL
LIN {X 0,Y 474.59,Z 546.788,A -85,B 0,C 180,E1 -14348.475,E2 -14348.475} C_VEL
LIN {X 0,Y 478.814,Z 480.116,A -85,B 0,C 180,E1 -14349.79,E2 -14349.79} C_VEL
LIN {X 0,Y 482.228,Z 404.363,A -85,B 0,C 180,E1 -14351.037,E2 -14351.037} C_VEL
LIN {X 0,Y 482.865,Z 388.766,A -85,B 0,C 180,E1 -14351.284,E2 -14351.284} C_VEL
LIN {X 0,Y 487.692,Z 367.209,A -85,B 0,C 180,E1 -14352.1,E2 -14352.1} C_VEL
LIN {X 0,Y 488.087,Z 337.279,A -85,B 0,C 180,E1 -14354.192,E2 -14354.192} C_VEL
LIN {X 0,Y 480.525,Z 316.786,A -85,B 0,C 180,E1 -14356.796,E2 -14356.796} C_VEL
LIN {X 0,Y 473.272,Z 299.429,A -85,B 0,C 180,E1 -14359.244,E2 -14359.244} C_VEL
LIN {X 0,Y 465.37,Z 283.001,A -85,B 0,C 180,E1 -14361.772,E2 -14361.772} C_VEL
LIN {X 0,Y 458.52,Z 270.201,A -85,B 0,C 180,E1 -14363.929,E2 -14363.929} C_VEL
LIN {X 0,Y 451.389,Z 257.758,A -85,B 0,C 180,E1 -14366.22,E2 -14366.22} C_VEL
LIN {X 0,Y 447.535,Z 251.832,A -85,B 0,C 180,E1 -14367.422,E2 -14367.422} C_VEL
LIN {X 0,Y 444.581,Z 247.118,A -85,B 0,C 180,E1 -14368.397,E2 -14368.397} C_VEL
LIN {X 0,Y 442.024,Z 242.9,A -85,B 0,C 180,E1 -14369.27,E2 -14369.27} C_VEL
LIN {X 0,Y 439.004,Z 238.993,A -85,B 0,C 180,E1 -14370.23,E2 -14370.23} C_VEL
LIN {X 0,Y 438.078,Z 236.858,A -85,B 0,C 180,E1 -14370.611,E2 -14370.611} C_VEL
LIN {X 0,Y 435.686,Z 234.524,A -85,B 0,C 180,E1 -14371.337,E2 -14371.337} C_VEL
LIN {X 0,Y 434.427,Z 231.152,A -85,B 0,C 180,E1 -14371.918,E2 -14371.918} C_VEL
LIN {X 0,Y 434.413,Z 231.077,A -85,B 0,C 180,E1 -14375.814,E2 -14375.814} C_VEL
LIN {X 0,Y 434.415,Z 231.111,A -85,B 0,C 180,E1 -14379.521,E2 -14379.521} C_VEL
LIN {X 0,Y 434.41,Z 231.082,A -85,B 0,C 180,E1 -14383.279,E2 -14383.279} C_VEL
LIN {X 0,Y 434.414,Z 231.07,A -85,B 0,C 180,E1 -14386.964,E2 -14386.964} C_VEL
LIN {X 0,Y 434.417,Z 231.117,A -85,B 0,C 180,E1 -14390.862,E2 -14390.862} C_VEL
LIN {X 0,Y 434.4,Z 231.067,A -85,B 0,C 180,E1 -14394.585,E2 -14394.585} C_VEL
LIN {X 0,Y 434.4,Z 231.102,A -85,B 0,C 180,E1 -14398.417,E2 -14398.417} C_VEL
LIN {X 0,Y 434.397,Z 231.086,A -85,B 0,C 180,E1 -14402.243,E2 -14402.243} C_VEL
LIN {X 0,Y 434.407,Z 231.074,A -85,B 0,C 180,E1 -14405.945,E2 -14405.945} C_VEL
LIN {X 0,Y 434.417,Z 231.109,A -85,B 0,C 180,E1 -14409.673,E2 -14409.673} C_VEL
LIN {X 0,Y 434.422,Z 231.116,A -85,B 0,C 180,E1 -14413.442,E2 -14413.442} C_VEL
LIN {X 0,Y 434.418,Z 231.119,A -85,B 0,C 180,E1 -14417.273,E2 -14417.273} C_VEL
LIN {X 0,Y 434.405,Z 231.11,A -85,B 0,C 180,E1 -14421.043,E2 -14421.043} C_VEL
LIN {X 0,Y 434.462,Z 231.349,A -85,B 0,C 180,E1 -14421.607,E2 -14421.607} C_VEL
LIN {X 0,Y 435.727,Z 234.638,A -85,B 0,C 180,E1 -14422.249,E2 -14422.249} C_VEL
LIN {X 0,Y 436.823,Z 236.057,A -85,B 0,C 180,E1 -14422.616,E2 -14422.616} C_VEL
LIN {X 0,Y 438.586,Z 239.757,A -85,B 0,C 180,E1 -14423.371,E2 -14423.371} C_VEL
LIN {X 0,Y 444.512,Z 251.087,A -85,B 0,C 180,E1 -14425.73,E2 -14425.73} C_VEL
LIN {X 0,Y 451.703,Z 264.954,A -85,B 0,C 180,E1 -14428.42,E2 -14428.42} C_VEL
LIN {X 0,Y 460.948,Z 283.156,A -85,B 0,C 180,E1 -14431.665,E2 -14431.665} C_VEL
LIN {X 0,Y 470.989,Z 303.713,A -85,B 0,C 180,E1 -14434.974,E2 -14434.974} C_VEL
LIN {X 0,Y 480.444,Z 323.416,A -85,B 0,C 180,E1 -14437.819,E2 -14437.819} C_VEL
LIN {X 0,Y 492.32,Z 342.331,A -85,B 0,C 180,E1 -14439.462,E2 -14439.462} C_VEL
LIN {X 0,Y 493.116,Z 353.729,A -85,B 0,C 180,E1 -14439.811,E2 -14439.811} C_VEL
LIN {X 0,Y 479.816,Z 597.99,A -85,B 0,C 180,E1 -14444.217,E2 -14444.217} C_VEL
LIN {X 0,Y 475.206,Z 693.32,A -85,B 0,C 180,E1 -14445.945,E2 -14445.945} C_VEL
LIN {X 0,Y 473.089,Z 717.844,A -85,B 0,C 180,E1 -14446.589,E2 -14446.589} C_VEL
LIN {X 0,Y 470.471,Z 742.347,A -85,B 0,C 180,E1 -14447.439,E2 -14447.439} C_VEL
LIN {X 0,Y 467.661,Z 764.279,A -85,B 0,C 180,E1 -14448.404,E2 -14448.404} C_VEL
LIN {X 0,Y 464.068,Z 788.83,A -85,B 0,C 180,E1 -14449.73,E2 -14449.73} C_VEL
LIN {X 0,Y 460.557,Z 810.563,A -85,B 0,C 180,E1 -14451.139,E2 -14451.139} C_VEL
LIN {X 0,Y 456.832,Z 831.454,A -85,B 0,C 180,E1 -14452.758,E2 -14452.758} C_VEL
LIN {X 0,Y 453.028,Z 851.892,A -85,B 0,C 180,E1 -14454.597,E2 -14454.597} C_VEL
LIN {X 0,Y 449.468,Z 870.25,A -85,B 0,C 180,E1 -14456.536,E2 -14456.536} C_VEL
LIN {X 0,Y 445.834,Z 888.842,A -85,B 0,C 180,E1 -14458.797,E2 -14458.797} C_VEL
LIN {X 0,Y 442.844,Z 904.158,A -85,B 0,C 180,E1 -14460.958,E2 -14460.958} C_VEL
LIN {X 0,Y 439.83,Z 920.376,A -85,B 0,C 180,E1 -14463.599,E2 -14463.599} C_VEL
LIN {X 0,Y 437.547,Z 933.458,A -85,B 0,C 180,E1 -14466.077,E2 -14466.077} C_VEL
LIN {X 0,Y 435.492,Z 946.713,A -85,B 0,C 180,E1 -14469.012,E2 -14469.012} C_VEL
LIN {X 0,Y 434.204,Z 956.661,A -85,B 0,C 180,E1 -14471.61,E2 -14471.61} C_VEL
LIN {X 0,Y 433.18,Z 966.726,A -85,B 0,C 180,E1 -14474.765,E2 -14474.765} C_VEL
LIN {X 0,Y 432.709,Z 973.704,A -85,B 0,C 180,E1 -14477.455,E2 -14477.455} C_VEL
LIN {X 0,Y 432.51,Z 980.015,A -85,B 0,C 180,E1 -14480.553,E2 -14480.553} C_VEL
LIN {X 0,Y 432.525,Z 983.969,A -85,B 0,C 180,E1 -14483.229,E2 -14483.229} C_VEL
LIN {X 0,Y 432.609,Z 986.642,A -85,B 0,C 180,E1 -14485.891,E2 -14485.891} C_VEL
LIN {X 0,Y 432.684,Z 988.026,A -85,B 0,C 180,E1 -14488.941,E2 -14488.941} C_VEL
LIN {X 0,Y 432.693,Z 987.865,A -85,B 0,C 180,E1 -14491.457,E2 -14491.457} C_VEL
LIN {X 0,Y 432.625,Z 986.465,A -85,B 0,C 180,E1 -14494.109,E2 -14494.109} C_VEL
LIN {X 0,Y 432.518,Z 983.402,A -85,B 0,C 180,E1 -14497.038,E2 -14497.038} C_VEL
LIN {X 0,Y 432.535,Z 978.948,A -85,B 0,C 180,E1 -14499.85,E2 -14499.85} C_VEL
LIN {X 0,Y 432.746,Z 972.775,A -85,B 0,C 180,E1 -14502.822,E2 -14502.822} C_VEL
LIN {X 0,Y 433.299,Z 964.787,A -85,B 0,C 180,E1 -14505.801,E2 -14505.801} C_VEL
LIN {X 0,Y 434.282,Z 955.593,A -85,B 0,C 180,E1 -14508.665,E2 -14508.665} C_VEL
LIN {X 0,Y 435.918,Z 943.785,A -85,B 0,C 180,E1 -14511.724,E2 -14511.724} C_VEL
LIN {X 0,Y 438.19,Z 930.428,A -85,B 0,C 180,E1 -14514.682,E2 -14514.682} C_VEL
LIN {X 0,Y 440.937,Z 915.903,A -85,B 0,C 180,E1 -14517.409,E2 -14517.409} C_VEL
LIN {X 0,Y 444.43,Z 899.316,A -85,B 0,C 180,E1 -14520.113,E2 -14520.113} C_VEL
LIN {X 0,Y 447.961,Z 883.142,A -85,B 0,C 180,E1 -14522.392,E2 -14522.392} C_VEL
LIN {X 0,Y 452.503,Z 863.23,A -85,B 0,C 180,E1 -14524.826,E2 -14524.826} C_VEL
LIN {X 0,Y 457.214,Z 842.793,A -85,B 0,C 180,E1 -14526.971,E2 -14526.971} C_VEL
LIN {X 0,Y 461.973,Z 821.362,A -85,B 0,C 180,E1 -14528.879,E2 -14528.879} C_VEL
LIN {X 0,Y 466.951,Z 798.439,A -85,B 0,C 180,E1 -14530.614,E2 -14530.614} C_VEL
LIN {X 0,Y 471.451,Z 776.7,A -85,B 0,C 180,E1 -14532.001,E2 -14532.001} C_VEL
LIN {X 0,Y 475.647,Z 754.482,A -85,B 0,C 180,E1 -14533.177,E2 -14533.177} C_VEL
LIN {X 0,Y 479.769,Z 730.807,A -85,B 0,C 180,E1 -14534.206,E2 -14534.206} C_VEL
LIN {X 0,Y 483.218,Z 708.005,A -85,B 0,C 180,E1 -14534.989,E2 -14534.989} C_VEL
LIN {X 0,Y 486.34,Z 682.731,A -85,B 0,C 180,E1 -14535.648,E2 -14535.648} C_VEL
LIN {X 0,Y 494.076,Z 612.481,A -85,B 0,C 180,E1 -14537.206,E2 -14537.206} C_VEL
LIN {X 0,Y 502.506,Z 553.906,A -85,B 0,C 180,E1 -14538.583,E2 -14538.583} C_VEL
LIN {X 0,Y 513.155,Z 495.233,A -85,B 0,C 180,E1 -14540.013,E2 -14540.013} C_VEL
LIN {X 0,Y 520.231,Z 462.048,A -85,B 0,C 180,E1 -14540.83,E2 -14540.83} C_VEL
LIN {X 0,Y 514.117,Z 487.384,A -85,B 0,C 180,E1 -14542.369,E2 -14542.369} C_VEL
LIN {X 0,Y 508.478,Z 516.377,A -85,B 0,C 180,E1 -14543.917,E2 -14543.917} C_VEL
LIN {X 0,Y 507.364,Z 522.401,A -85,B 0,C 180,E1 -14544.175,E2 -14544.175} C_VEL
LIN {X 0,Y 487.121,Z 627.358,A -85,B 0,C 180,E1 -14547.257,E2 -14547.257} C_VEL
LIN {X 0,Y 475.859,Z 693.759,A -85,B 0,C 180,E1 -14549.349,E2 -14549.349} C_VEL
LIN {X 0,Y 471.445,Z 717.142,A -85,B 0,C 180,E1 -14550.315,E2 -14550.315} C_VEL
LIN {X 0,Y 466.821,Z 740.453,A -85,B 0,C 180,E1 -14551.538,E2 -14551.538} C_VEL
LIN {X 0,Y 462.255,Z 762.889,A -85,B 0,C 180,E1 -14552.983,E2 -14552.983} C_VEL
LIN {X 0,Y 457.972,Z 783.621,A -85,B 0,C 180,E1 -14554.595,E2 -14554.595} C_VEL
LIN {X 0,Y 454.035,Z 802.687,A -85,B 0,C 180,E1 -14556.371,E2 -14556.371} C_VEL
LIN {X 0,Y 450.491,Z 819.554,A -85,B 0,C 180,E1 -14558.243,E2 -14558.243} C_VEL
LIN {X 0,Y 447.216,Z 834.742,A -85,B 0,C 180,E1 -14560.269,E2 -14560.269} C_VEL
LIN {X 0,Y 444.24,Z 848.199,A -85,B 0,C 180,E1 -14562.446,E2 -14562.446} C_VEL
LIN {X 0,Y 441.869,Z 858.654,A -85,B 0,C 180,E1 -14564.513,E2 -14564.513} C_VEL
LIN {X 0,Y 439.826,Z 867.472,A -85,B 0,C 180,E1 -14566.657,E2 -14566.657} C_VEL
LIN {X 0,Y 437.956,Z 875.128,A -85,B 0,C 180,E1 -14569.077,E2 -14569.077} C_VEL
LIN {X 0,Y 436.551,Z 880.519,A -85,B 0,C 180,E1 -14571.438,E2 -14571.438} C_VEL
LIN {X 0,Y 435.506,Z 884.037,A -85,B 0,C 180,E1 -14573.805,E2 -14573.805} C_VEL
LIN {X 0,Y 434.739,Z 885.709,A -85,B 0,C 180,E1 -14576.176,E2 -14576.176} C_VEL
LIN {X 0,Y 434.252,Z 885.662,A -85,B 0,C 180,E1 -14578.417,E2 -14578.417} C_VEL
LIN {X 0,Y 433.949,Z 883.916,A -85,B 0,C 180,E1 -14580.792,E2 -14580.792} C_VEL
LIN {X 0,Y 433.822,Z 880.414,A -85,B 0,C 180,E1 -14583.171,E2 -14583.171} C_VEL
LIN {X 0,Y 433.898,Z 875.128,A -85,B 0,C 180,E1 -14585.554,E2 -14585.554} C_VEL
LIN {X 0,Y 434.191,Z 867.946,A -85,B 0,C 180,E1 -14587.942,E2 -14587.942} C_VEL
LIN {X 0,Y 434.752,Z 858.696,A -85,B 0,C 180,E1 -14590.334,E2 -14590.334} C_VEL
LIN {X 0,Y 435.588,Z 847.848,A -85,B 0,C 180,E1 -14592.596,E2 -14592.596} C_VEL
LIN {X 0,Y 436.677,Z 835.492,A -85,B 0,C 180,E1 -14594.724,E2 -14594.724} C_VEL
LIN {X 0,Y 438.002,Z 821.663,A -85,B 0,C 180,E1 -14596.717,E2 -14596.717} C_VEL
LIN {X 0,Y 439.526,Z 806.355,A -85,B 0,C 180,E1 -14598.572,E2 -14598.572} C_VEL
LIN {X 0,Y 441.297,Z 788.852,A -85,B 0,C 180,E1 -14600.353,E2 -14600.353} C_VEL
LIN {X 0,Y 443.116,Z 770.098,A -85,B 0,C 180,E1 -14601.936,E2 -14601.936} C_VEL
LIN {X 0,Y 444.956,Z 750.504,A -85,B 0,C 180,E1 -14603.297,E2 -14603.297} C_VEL
LIN {X 0,Y 446.74,Z 729.864,A -85,B 0,C 180,E1 -14604.461,E2 -14604.461} C_VEL
LIN {X 0,Y 448.439,Z 707.503,A -85,B 0,C 180,E1 -14605.448,E2 -14605.448} C_VEL
LIN {X 0,Y 449.902,Z 685.211,A -85,B 0,C 180,E1 -14606.178,E2 -14606.178} C_VEL
LIN {X 0,Y 458.982,Z 504.432,A -85,B 0,C 180,E1 -14610.184,E2 -14610.184} C_VEL
LIN {X 0,Y 453.98,Z 440.307,A -85,B 0,C 180,E1 -14612.209,E2 -14612.209} C_VEL
LIN {X 0,Y 459.668,Z 389.317,A -85,B 0,C 180,E1 -14616.276,E2 -14616.276} C_VEL
LIN {X 0,Y 465.95,Z 337.928,A -85,B 0,C 180,E1 -14620.396,E2 -14620.396} C_VEL
LIN {X 0,Y 468.304,Z 320.279,A -85,B 0,C 180,E1 -14621.813,E2 -14621.813} C_VEL
LIN {X 0,Y 469.999,Z 320.421,A -85,B 0,C 180,E1 -14622.078,E2 -14622.078} C_VEL
LIN {X 0,Y 472.95,Z 319.101,A -85,B 0,C 180,E1 -14622.409,E2 -14622.409} C_VEL
LIN {X 0,Y 473.758,Z 318.551,A -85,B 0,C 180,E1 -14622.484,E2 -14622.484} C_VEL
LIN {X 0,Y 481.12,Z 318.541,A -85,B 0,C 180,E1 -14623.547,E2 -14623.547} C_VEL
LIN {X 0,Y 488.11,Z 337.655,A -85,B 0,C 180,E1 -14625.953,E2 -14625.953} C_VEL
LIN {X 0,Y 487.583,Z 367.186,A -85,B 0,C 180,E1 -14628.003,E2 -14628.003} C_VEL
LIN {X 0,Y 482.724,Z 389.849,A -85,B 0,C 180,E1 -14628.836,E2 -14628.836} C_VEL
LIN {X 0,Y 479.12,Z 473.033,A -85,B 0,C 180,E1 -14630.183,E2 -14630.183} C_VEL
LIN {X 0,Y 475.182,Z 537.396,A -85,B 0,C 180,E1 -14631.427,E2 -14631.427} C_VEL
LIN {X 0,Y 469.914,Z 606.927,A -85,B 0,C 180,E1 -14632.993,E2 -14632.993} C_VEL
LIN {X 0,Y 466.667,Z 651.872,A -85,B 0,C 180,E1 -14634.173,E2 -14634.173} C_VEL
LIN {X 0,Y 465.17,Z 673.986,A -85,B 0,C 180,E1 -14634.915,E2 -14634.915} C_VEL
LIN {X 0,Y 463.302,Z 694.051,A -85,B 0,C 180,E1 -14635.791,E2 -14635.791} C_VEL
LIN {X 0,Y 463.124,Z 695.785,A -85,B 0,C 180,E1 -14635.876,E2 -14635.876} C_VEL
LIN {X 0,Y 461.533,Z 703.006,A -85,B 0,C 180,E1 -14636.171,E2 -14636.171} C_VEL
LIN {X 0,Y 454.331,Z 721.147,A -85,B 0,C 180,E1 -14636.792,E2 -14636.792} C_VEL
LIN {X 0,Y 452.526,Z 727.999,A -85,B 0,C 180,E1 -14637.18,E2 -14637.18} C_VEL
LIN {X 0,Y 449.433,Z 747.73,A -85,B 0,C 180,E1 -14638.685,E2 -14638.685} C_VEL
LIN {X 0,Y 446.115,Z 766.61,A -85,B 0,C 180,E1 -14640.417,E2 -14640.417} C_VEL
LIN {X 0,Y 442.734,Z 784.281,A -85,B 0,C 180,E1 -14642.347,E2 -14642.347} C_VEL
LIN {X 0,Y 439.536,Z 800.082,A -85,B 0,C 180,E1 -14644.391,E2 -14644.391} C_VEL
LIN {X 0,Y 436.629,Z 814.087,A -85,B 0,C 180,E1 -14646.518,E2 -14646.518} C_VEL
LIN {X 0,Y 433.818,Z 827.523,A -85,B 0,C 180,E1 -14648.927,E2 -14648.927} C_VEL
LIN {X 0,Y 431.257,Z 840.011,A -85,B 0,C 180,E1 -14651.62,E2 -14651.62} C_VEL
LIN {X 0,Y 429.163,Z 850.783,A -85,B 0,C 180,E1 -14654.459,E2 -14654.459} C_VEL
LIN {X 0,Y 427.642,Z 859.422,A -85,B 0,C 180,E1 -14657.303,E2 -14657.303} C_VEL
LIN {X 0,Y 426.613,Z 865.849,A -85,B 0,C 180,E1 -14660.012,E2 -14660.012} C_VEL
LIN {X 0,Y 425.948,Z 870.878,A -85,B 0,C 180,E1 -14662.853,E2 -14662.853} C_VEL
LIN {X 0,Y 425.573,Z 874.236,A -85,B 0,C 180,E1 -14665.688,E2 -14665.688} C_VEL
LIN {X 0,Y 425.411,Z 875.978,A -85,B 0,C 180,E1 -14668.518,E2 -14668.518} C_VEL
LIN {X 0,Y 425.396,Z 876.037,A -85,B 0,C 180,E1 -14671.212,E2 -14671.212} C_VEL
LIN {X 0,Y 425.541,Z 874.534,A -85,B 0,C 180,E1 -14674.042,E2 -14674.042} C_VEL
LIN {X 0,Y 425.89,Z 871.42,A -85,B 0,C 180,E1 -14676.877,E2 -14676.877} C_VEL
LIN {X 0,Y 426.517,Z 866.643,A -85,B 0,C 180,E1 -14679.717,E2 -14679.717} C_VEL
LIN {X 0,Y 427.548,Z 860.065,A -85,B 0,C 180,E1 -14682.562,E2 -14682.562} C_VEL
LIN {X 0,Y 429.023,Z 851.551,A -85,B 0,C 180,E1 -14685.408,E2 -14685.408} C_VEL
LIN {X 0,Y 430.845,Z 842.034,A -85,B 0,C 180,E1 -14687.979,E2 -14687.979} C_VEL
LIN {X 0,Y 433.169,Z 830.622,A -85,B 0,C 180,E1 -14690.54,E2 -14690.54} C_VEL
LIN {X 0,Y 436.027,Z 817.006,A -85,B 0,C 180,E1 -14693.087,E2 -14693.087} C_VEL
LIN {X 0,Y 439.047,Z 802.603,A -85,B 0,C 180,E1 -14695.35,E2 -14695.35} C_VEL
LIN {X 0,Y 442.22,Z 787.088,A -85,B 0,C 180,E1 -14697.417,E2 -14697.417} C_VEL
LIN {X 0,Y 445.46,Z 770.482,A -85,B 0,C 180,E1 -14699.296,E2 -14699.296} C_VEL
LIN {X 0,Y 448.778,Z 752.101,A -85,B 0,C 180,E1 -14701.05,E2 -14701.05} C_VEL
LIN {X 0,Y 451.954,Z 732.415,A -85,B 0,C 180,E1 -14702.616,E2 -14702.616} C_VEL
LIN {X 0,Y 454.795,Z 712.053,A -85,B 0,C 180,E1 -14703.947,E2 -14703.947} C_VEL
LIN {X 0,Y 457.165,Z 691.454,A -85,B 0,C 180,E1 -14705.039,E2 -14705.039} C_VEL
LIN {X 0,Y 459.051,Z 670.445,A -85,B 0,C 180,E1 -14705.917,E2 -14705.917} C_VEL
LIN {X 0,Y 460.847,Z 643.521,A -85,B 0,C 180,E1 -14706.762,E2 -14706.762} C_VEL
LIN {X 0,Y 465.018,Z 591.098,A -85,B 0,C 180,E1 -14708.101,E2 -14708.101} C_VEL
LIN {X 0,Y 469.955,Z 525.918,A -85,B 0,C 180,E1 -14709.541,E2 -14709.541} C_VEL
LIN {X 0,Y 473.829,Z 460.766,A -85,B 0,C 180,E1 -14710.769,E2 -14710.769} C_VEL
LIN {X 0,Y 476.944,Z 390.939,A -85,B 0,C 180,E1 -14711.906,E2 -14711.906} C_VEL
LIN {X 0,Y 481.922,Z 368.425,A -85,B 0,C 180,E1 -14712.764,E2 -14712.764} C_VEL
LIN {X 0,Y 482.284,Z 341.272,A -85,B 0,C 180,E1 -14714.673,E2 -14714.673} C_VEL
LIN {X 0,Y 474.795,Z 320.884,A -85,B 0,C 180,E1 -14717.303,E2 -14717.303} C_VEL
LIN {X 0,Y 467.967,Z 304.452,A -85,B 0,C 180,E1 -14719.653,E2 -14719.653} C_VEL
LIN {X 0,Y 459.483,Z 286.611,A -85,B 0,C 180,E1 -14722.46,E2 -14722.46} C_VEL
LIN {X 0,Y 451.665,Z 272.099,A -85,B 0,C 180,E1 -14725.014,E2 -14725.014} C_VEL
LIN {X 0,Y 444.206,Z 259.342,A -85,B 0,C 180,E1 -14727.454,E2 -14727.454} C_VEL
LIN {X 0,Y 440.149,Z 253.195,A -85,B 0,C 180,E1 -14728.805,E2 -14728.805} C_VEL
LIN {X 0,Y 437.232,Z 248.646,A -85,B 0,C 180,E1 -14729.794,E2 -14729.794} C_VEL
LIN {X 0,Y 434.72,Z 244.895,A -85,B 0,C 180,E1 -14730.665,E2 -14730.665} C_VEL
LIN {X 0,Y 434.076,Z 243.594,A -85,B 0,C 180,E1 -14730.919,E2 -14730.919} C_VEL
LIN {X 0,Y 431.481,Z 240.519,A -85,B 0,C 180,E1 -14731.788,E2 -14731.788} C_VEL
LIN {X 0,Y 430.122,Z 237.835,A -85,B 0,C 180,E1 -14732.337,E2 -14732.337} C_VEL
LIN {X 0,Y 427.62,Z 235.33,A -85,B 0,C 180,E1 -14733.174,E2 -14733.174} C_VEL
LIN {X 0,Y 426.48,Z 232.123,A -85,B 0,C 180,E1 -14733.739,E2 -14733.739} C_VEL
LIN {X 0,Y 426.481,Z 232.07,A -85,B 0,C 180,E1 -14737.678,E2 -14737.678} C_VEL
LIN {X 0,Y 426.472,Z 232.056,A -85,B 0,C 180,E1 -14741.548,E2 -14741.548} C_VEL
LIN {X 0,Y 426.474,Z 232.097,A -85,B 0,C 180,E1 -14745.332,E2 -14745.332} C_VEL
LIN {X 0,Y 426.473,Z 232.069,A -85,B 0,C 180,E1 -14749.225,E2 -14749.225} C_VEL
LIN {X 0,Y 426.483,Z 232.059,A -85,B 0,C 180,E1 -14752.997,E2 -14752.997} C_VEL
LIN {X 0,Y 426.472,Z 232.107,A -85,B 0,C 180,E1 -14756.909,E2 -14756.909} C_VEL
LIN {X 0,Y 426.46,Z 232.051,A -85,B 0,C 180,E1 -14760.672,E2 -14760.672} C_VEL
LIN {X 0,Y 426.46,Z 232.102,A -85,B 0,C 180,E1 -14764.572,E2 -14764.572} C_VEL
LIN {X 0,Y 426.452,Z 232.062,A -85,B 0,C 180,E1 -14768.359,E2 -14768.359} C_VEL
LIN {X 0,Y 426.462,Z 232.111,A -85,B 0,C 180,E1 -14772.182,E2 -14772.182} C_VEL
LIN {X 0,Y 426.468,Z 232.097,A -85,B 0,C 180,E1 -14775.996,E2 -14775.996} C_VEL
LIN {X 0,Y 426.476,Z 232.108,A -85,B 0,C 180,E1 -14779.874,E2 -14779.874} C_VEL
LIN {X 0,Y 426.478,Z 232.265,A -85,B 0,C 180,E1 -14780.272,E2 -14780.272} C_VEL
LIN {X 0,Y 427.763,Z 235.579,A -85,B 0,C 180,E1 -14780.955,E2 -14780.955} C_VEL
LIN {X 0,Y 429.097,Z 237.552,A -85,B 0,C 180,E1 -14781.46,E2 -14781.46} C_VEL
LIN {X 0,Y 430.846,Z 241.073,A -85,B 0,C 180,E1 -14782.228,E2 -14782.228} C_VEL
LIN {X 0,Y 436.457,Z 251.678,A -85,B 0,C 180,E1 -14784.498,E2 -14784.498} C_VEL
LIN {X 0,Y 443.835,Z 266.001,A -85,B 0,C 180,E1 -14787.36,E2 -14787.36} C_VEL
LIN {X 0,Y 452.566,Z 283.268,A -85,B 0,C 180,E1 -14790.541,E2 -14790.541} C_VEL
LIN {X 0,Y 462.107,Z 302.657,A -85,B 0,C 180,E1 -14793.786,E2 -14793.786} C_VEL
LIN {X 0,Y 472.195,Z 323.815,A -85,B 0,C 180,E1 -14796.969,E2 -14796.969} C_VEL
LIN {X 0,Y 486.355,Z 346.135,A -85,B 0,C 180,E1 -14798.965,E2 -14798.965} C_VEL
LIN {X 0,Y 486.887,Z 355.043,A -85,B 0,C 180,E1 -14799.235,E2 -14799.235} C_VEL
LIN {X 0,Y 473.101,Z 598.027,A -85,B 0,C 180,E1 -14803.694,E2 -14803.694} C_VEL
LIN {X 0,Y 468.309,Z 693.219,A -85,B 0,C 180,E1 -14805.451,E2 -14805.451} C_VEL
LIN {X 0,Y 466.145,Z 717.602,A -85,B 0,C 180,E1 -14806.101,E2 -14806.101} C_VEL
LIN {X 0,Y 463.515,Z 741.606,A -85,B 0,C 180,E1 -14806.941,E2 -14806.941} C_VEL
LIN {X 0,Y 460.717,Z 762.87,A -85,B 0,C 180,E1 -14807.885,E2 -14807.885} C_VEL
LIN {X 0,Y 457.151,Z 786.865,A -85,B 0,C 180,E1 -14809.181,E2 -14809.181} C_VEL
LIN {X 0,Y 453.657,Z 807.865,A -85,B 0,C 180,E1 -14810.548,E2 -14810.548} C_VEL
LIN {X 0,Y 449.741,Z 829.66,A -85,B 0,C 180,E1 -14812.229,E2 -14812.229} C_VEL
LIN {X 0,Y 445.89,Z 849.884,A -85,B 0,C 180,E1 -14814.05,E2 -14814.05} C_VEL
LIN {X 0,Y 442.14,Z 868.681,A -85,B 0,C 180,E1 -14816.042,E2 -14816.042} C_VEL
LIN {X 0,Y 438.483,Z 886.955,A -85,B 0,C 180,E1 -14818.274,E2 -14818.274} C_VEL
LIN {X 0,Y 435.26,Z 902.953,A -85,B 0,C 180,E1 -14820.554,E2 -14820.554} C_VEL
LIN {X 0,Y 432.19,Z 918.993,A -85,B 0,C 180,E1 -14823.183,E2 -14823.183} C_VEL
LIN {X 0,Y 429.947,Z 931.377,A -85,B 0,C 180,E1 -14825.546,E2 -14825.546} C_VEL
LIN {X 0,Y 427.893,Z 944.08,A -85,B 0,C 180,E1 -14828.333,E2 -14828.333} C_VEL
LIN {X 0,Y 426.398,Z 954.751,A -85,B 0,C 180,E1 -14831.119,E2 -14831.119} C_VEL
LIN {X 0,Y 425.364,Z 964.265,A -85,B 0,C 180,E1 -14834.036,E2 -14834.036} C_VEL
LIN {X 0,Y 424.793,Z 972.078,A -85,B 0,C 180,E1 -14837.031,E2 -14837.031} C_VEL
LIN {X 0,Y 424.553,Z 978.232,A -85,B 0,C 180,E1 -14839.963,E2 -14839.963} C_VEL
LIN {X 0,Y 424.551,Z 982.756,A -85,B 0,C 180,E1 -14842.965,E2 -14842.965} C_VEL
LIN {X 0,Y 424.647,Z 985.404,A -85,B 0,C 180,E1 -14845.544,E2 -14845.544} C_VEL
LIN {X 0,Y 424.735,Z 987.033,A -85,B 0,C 180,E1 -14848.516,E2 -14848.516} C_VEL
LIN {X 0,Y 424.748,Z 986.967,A -85,B 0,C 180,E1 -14851.349,E2 -14851.349} C_VEL
LIN {X 0,Y 424.675,Z 985.626,A -85,B 0,C 180,E1 -14854.051,E2 -14854.051} C_VEL
LIN {X 0,Y 424.549,Z 982.683,A -85,B 0,C 180,E1 -14857.035,E2 -14857.035} C_VEL
LIN {X 0,Y 424.556,Z 978.274,A -85,B 0,C 180,E1 -14859.9,E2 -14859.9} C_VEL
LIN {X 0,Y 424.75,Z 972.469,A -85,B 0,C 180,E1 -14862.784,E2 -14862.784} C_VEL
LIN {X 0,Y 425.336,Z 964.289,A -85,B 0,C 180,E1 -14865.965,E2 -14865.965} C_VEL
LIN {X 0,Y 426.303,Z 955.621,A -85,B 0,C 180,E1 -14868.744,E2 -14868.744} C_VEL
LIN {X 0,Y 428.057,Z 943.596,A -85,B 0,C 180,E1 -14871.975,E2 -14871.975} C_VEL
LIN {X 0,Y 430.2,Z 931.534,A -85,B 0,C 180,E1 -14874.731,E2 -14874.731} C_VEL
LIN {X 0,Y 433.18,Z 916.69,A -85,B 0,C 180,E1 -14877.643,E2 -14877.643} C_VEL
LIN {X 0,Y 436.804,Z 900.467,A -85,B 0,C 180,E1 -14880.391,E2 -14880.391} C_VEL
LIN {X 0,Y 440.698,Z 883.603,A -85,B 0,C 180,E1 -14882.838,E2 -14882.838} C_VEL
LIN {X 0,Y 445.139,Z 865.398,A -85,B 0,C 180,E1 -14885.151,E2 -14885.151} C_VEL
LIN {X 0,Y 449.915,Z 845.746,A -85,B 0,C 180,E1 -14887.286,E2 -14887.286} C_VEL
LIN {X 0,Y 455.25,Z 823.443,A -85,B 0,C 180,E1 -14889.365,E2 -14889.365} C_VEL
LIN {X 0,Y 460.376,Z 801.638,A -85,B 0,C 180,E1 -14891.092,E2 -14891.092} C_VEL
LIN {X 0,Y 465.154,Z 780.008,A -85,B 0,C 180,E1 -14892.525,E2 -14892.525} C_VEL
LIN {X 0,Y 470.242,Z 755.462,A -85,B 0,C 180,E1 -14893.883,E2 -14893.883} C_VEL
LIN {X 0,Y 474.678,Z 732.122,A -85,B 0,C 180,E1 -14894.93,E2 -14894.93} C_VEL
LIN {X 0,Y 478.408,Z 709.551,A -85,B 0,C 180,E1 -14895.731,E2 -14895.731} C_VEL
LIN {X 0,Y 482.08,Z 683.101,A -85,B 0,C 180,E1 -14896.45,E2 -14896.45} C_VEL
LIN {X 0,Y 490.399,Z 615.868,A -85,B 0,C 180,E1 -14897.988,E2 -14897.988} C_VEL
LIN {X 0,Y 499.619,Z 558.231,A -85,B 0,C 180,E1 -14899.37,E2 -14899.37} C_VEL
LIN {X 0,Y 510.732,Z 502.233,A -85,B 0,C 180,E1 -14900.747,E2 -14900.747} C_VEL
LIN {X 0,Y 514.736,Z 484.385,A -85,B 0,C 180,E1 -14901.201,E2 -14901.201} C_VEL
LIN {X 0,Y 508.019,Z 513.092,A -85,B 0,C 180,E1 -14902.781,E2 -14902.781} C_VEL
LIN {X 0,Y 505.729,Z 524.168,A -85,B 0,C 180,E1 -14903.311,E2 -14903.311} C_VEL
LIN {X 0,Y 484.235,Z 628.309,A -85,B 0,C 180,E1 -14906.382,E2 -14906.382} C_VEL
LIN {X 0,Y 472.206,Z 693.862,A -85,B 0,C 180,E1 -14908.474,E2 -14908.474} C_VEL
LIN {X 0,Y 467.335,Z 717.432,A -85,B 0,C 180,E1 -14909.459,E2 -14909.459} C_VEL
LIN {X 0,Y 462.141,Z 741.15,A -85,B 0,C 180,E1 -14910.727,E2 -14910.727} C_VEL
LIN {X 0,Y 457.024,Z 763.873,A -85,B 0,C 180,E1 -14912.224,E2 -14912.224} C_VEL
LIN {X 0,Y 452.238,Z 784.865,A -85,B 0,C 180,E1 -14913.897,E2 -14913.897} C_VEL
LIN {X 0,Y 447.854,Z 804.185,A -85,B 0,C 180,E1 -14915.745,E2 -14915.745} C_VEL
LIN {X 0,Y 443.79,Z 821.736,A -85,B 0,C 180,E1 -14917.758,E2 -14917.758} C_VEL
LIN {X 0,Y 440.509,Z 835.783,A -85,B 0,C 180,E1 -14919.678,E2 -14919.678} C_VEL
LIN {X 0,Y 437.482,Z 848.495,A -85,B 0,C 180,E1 -14921.752,E2 -14921.752} C_VEL
LIN {X 0,Y 434.746,Z 859.667,A -85,B 0,C 180,E1 -14923.979,E2 -14923.979} C_VEL
LIN {X 0,Y 432.329,Z 869.151,A -85,B 0,C 180,E1 -14926.355,E2 -14926.355} C_VEL
LIN {X 0,Y 430.476,Z 876.136,A -85,B 0,C 180,E1 -14928.613,E2 -14928.613} C_VEL
LIN {X 0,Y 428.936,Z 881.586,A -85,B 0,C 180,E1 -14931.015,E2 -14931.015} C_VEL
LIN {X 0,Y 427.775,Z 885.109,A -85,B 0,C 180,E1 -14933.423,E2 -14933.423} C_VEL
LIN {X 0,Y 426.964,Z 886.798,A -85,B 0,C 180,E1 -14935.702,E2 -14935.702} C_VEL
LIN {X 0,Y 426.376,Z 886.86,A -85,B 0,C 180,E1 -14938.119,E2 -14938.119} C_VEL
LIN {X 0,Y 426.029,Z 885.173,A -85,B 0,C 180,E1 -14940.538,E2 -14940.538} C_VEL
LIN {X 0,Y 425.876,Z 881.732,A -85,B 0,C 180,E1 -14942.961,E2 -14942.961} C_VEL
LIN {X 0,Y 425.933,Z 876.496,A -85,B 0,C 180,E1 -14945.388,E2 -14945.388} C_VEL
LIN {X 0,Y 426.194,Z 869.835,A -85,B 0,C 180,E1 -14947.685,E2 -14947.685} C_VEL
LIN {X 0,Y 426.693,Z 861.334,A -85,B 0,C 180,E1 -14949.986,E2 -14949.986} C_VEL
LIN {X 0,Y 427.493,Z 850.799,A -85,B 0,C 180,E1 -14952.289,E2 -14952.289} C_VEL
LIN {X 0,Y 428.563,Z 838.672,A -85,B 0,C 180,E1 -14954.477,E2 -14954.477} C_VEL
LIN {X 0,Y 429.957,Z 824.273,A -85,B 0,C 180,E1 -14956.638,E2 -14956.638} C_VEL
LIN {X 0,Y 431.592,Z 808.256,A -85,B 0,C 180,E1 -14958.646,E2 -14958.646} C_VEL
LIN {X 0,Y 433.399,Z 790.898,A -85,B 0,C 180,E1 -14960.465,E2 -14960.465} C_VEL
LIN {X 0,Y 435.327,Z 771.859,A -85,B 0,C 180,E1 -14962.129,E2 -14962.129} C_VEL
LIN {X 0,Y 437.202,Z 752.517,A -85,B 0,C 180,E1 -14963.514,E2 -14963.514} C_VEL
LIN {X 0,Y 439.035,Z 732.107,A -85,B 0,C 180,E1 -14964.703,E2 -14964.703} C_VEL
LIN {X 0,Y 440.764,Z 710.262,A -85,B 0,C 180,E1 -14965.708,E2 -14965.708} C_VEL
LIN {X 0,Y 442.336,Z 687.29,A -85,B 0,C 180,E1 -14966.498,E2 -14966.498} C_VEL
LIN {X 0,Y 444.209,Z 649.813,A -85,B 0,C 180,E1 -14967.385,E2 -14967.385} C_VEL
LIN {X 0,Y 451.821,Z 505.144,A -85,B 0,C 180,E1 -14970.633,E2 -14970.633} C_VEL
LIN {X 0,Y 446.865,Z 439.5,A -85,B 0,C 180,E1 -14972.751,E2 -14972.751} C_VEL
LIN {X 0,Y 452.749,Z 388.876,A -85,B 0,C 180,E1 -14976.842,E2 -14976.842} C_VEL
LIN {X 0,Y 459.417,Z 336.523,A -85,B 0,C 180,E1 -14981.093,E2 -14981.093} C_VEL
LIN {X 0,Y 460.11,Z 332.118,A -85,B 0,C 180,E1 -14981.469,E2 -14981.469} C_VEL
LIN {X 0,Y 462.16,Z 332.055,A -85,B 0,C 180,E1 -14981.787,E2 -14981.787} C_VEL
